       // Index 3
       IF "HMI_Interface_Overview".homeCodition[3].pageIndex = 3 THEN
           "HMI_Interface_Overview".homeCodition[3].emOverviewTitle := WSTRING#'Attachment Home Condition 1';
           "HMI_Interface_Overview".homeCodition[3].emOverviewCmName[0] := WSTRING#'Top Tape X-Axis';
           "HMI_Interface_Overview".homeCodition[3].emOverviewCmName[1] := WSTRING#'Top Tape Attachment';
           "HMI_Interface_Overview".homeCodition[3].emOverviewCmName[2] := WSTRING#'Top Tape Attachment Vacuum';
           "HMI_Interface_Overview".homeCodition[3].emOverviewCmName[3] := WSTRING#'Spare';
           "HMI_Interface_Overview".homeCodition[3].emOverviewCmName[4] := WSTRING#'Spare';
           "HMI_Interface_Overview".homeCodition[3].emOverviewCmName[5] := WSTRING#'Spare';
           "HMI_Interface_Overview".homeCodition[3].emOverviewCmName[6] := WSTRING#'Spare';
           "HMI_Interface_Overview".homeCodition[3].emOverviewCmName[7] := WSTRING#'Spare';
           "HMI_Interface_Overview".homeCodition[3].emOverviewCmName[8] := WSTRING#'Spare';
           "HMI_Interface_Overview".homeCodition[3].emOverviewCmName[9] := WSTRING#'Spare';
           "HMI_Interface_Overview".homeCodition[3].emOverviewCmName[10] := WSTRING#'Spare';
           "HMI_Interface_Overview".homeCodition[3].emOverviewCmName[11] := WSTRING#'Spare';
           "HMI_Interface_Overview".homeCodition[3].emOverviewCmName[12] := WSTRING#'Spare';
           "HMI_Interface_Overview".homeCodition[3].emOverviewCmName[13] := WSTRING#'Spare';
           "HMI_Interface_Overview".homeCodition[3].emOverviewCmPositionName[0] := WSTRING#'Wait Position';
           "HMI_Interface_Overview".homeCodition[3].emOverviewCmPositionName[1] := WSTRING#'Up';
           "HMI_Interface_Overview".homeCodition[3].emOverviewCmPositionName[2] := WSTRING#'On';
           "HMI_Interface_Overview".homeCodition[3].emOverviewCmPositionName[3] := WSTRING#'Spare';
           "HMI_Interface_Overview".homeCodition[3].emOverviewCmPositionName[4] := WSTRING#'Spare';
           "HMI_Interface_Overview".homeCodition[3].emOverviewCmPositionName[5] := WSTRING#'Spare';
           "HMI_Interface_Overview".homeCodition[3].emOverviewCmPositionName[6] := WSTRING#'Spare';
           "HMI_Interface_Overview".homeCodition[3].emOverviewCmPositionName[7] := WSTRING#'Spare';
           "HMI_Interface_Overview".homeCodition[3].emOverviewCmPositionName[8] := WSTRING#'Spare';
           "HMI_Interface_Overview".homeCodition[3].emOverviewCmPositionName[9] := WSTRING#'Spare';
           "HMI_Interface_Overview".homeCodition[3].emOverviewCmPositionName[10] := WSTRING#'Spare';
           "HMI_Interface_Overview".homeCodition[3].emOverviewCmPositionName[11] := WSTRING#'Spare';
           "HMI_Interface_Overview".homeCodition[3].emOverviewCmPositionName[12] := WSTRING#'Spare';
           "HMI_Interface_Overview".homeCodition[3].emOverviewCmPositionName[13] := WSTRING#'Spare';
           IF NOT #statLampControl THEN
               "HMI_Interface_Overview".homeCodition[3].emOverviewHomeLampOn[0] := "Unit1.Em3.HmiInterface".cm.softcam.topTapeAxisX.pos00_wait.inPos;
               "HMI_Interface_Overview".homeCodition[3].emOverviewHomeLampOn[1] := "Unit1.Em3.HmiInterface".cmTopTapeAttachmentUpDown.monitoring.inHomePos;
               "HMI_Interface_Overview".homeCodition[3].emOverviewHomeLampOn[2] := "Unit1.Em3.HmiInterface".cmTopTapeAttachmentVaccumOffOn.monitoring.inWorkPos;
               "HMI_Interface_Overview".homeCodition[3].emOverviewHomeLampOn[3] := FALSE;
               "HMI_Interface_Overview".homeCodition[3].emOverviewHomeLampOn[4] := FALSE;
               "HMI_Interface_Overview".homeCodition[3].emOverviewHomeLampOn[5] := FALSE;
               "HMI_Interface_Overview".homeCodition[3].emOverviewHomeLampOn[6] := FALSE;
               "HMI_Interface_Overview".homeCodition[3].emOverviewHomeLampOn[7] := FALSE;
               "HMI_Interface_Overview".homeCodition[3].emOverviewHomeLampOn[8] := FALSE;
               "HMI_Interface_Overview".homeCodition[3].emOverviewHomeLampOn[9] := FALSE;
               "HMI_Interface_Overview".homeCodition[3].emOverviewHomeLampOn[10] := FALSE;
               "HMI_Interface_Overview".homeCodition[3].emOverviewHomeLampOn[11] := FALSE;
               "HMI_Interface_Overview".homeCodition[3].emOverviewHomeLampOn[12] := FALSE;
               "HMI_Interface_Overview".homeCodition[3].emOverviewHomeLampOn[13] := FALSE;
           END_IF;
       END_IF;

       // Index 4
       IF "HMI_Interface_Overview".homeCodition[3].pageIndex = 4 THEN
           "HMI_Interface_Overview".homeCodition[3].emOverviewTitle := WSTRING#'Fix Stage Home Condition 0';
           "HMI_Interface_Overview".homeCodition[3].emOverviewCmName[0] := WSTRING#'Top Tape Y-Axis';
           "HMI_Interface_Overview".homeCodition[3].emOverviewCmName[1] := WSTRING#'Top Tape Clamp Top Left';
           "HMI_Interface_Overview".homeCodition[3].emOverviewCmName[2] := WSTRING#'Top Tape Clamp Top Center';
           "HMI_Interface_Overview".homeCodition[3].emOverviewCmName[3] := WSTRING#'Top Tape Clamp Top Right';
           "HMI_Interface_Overview".homeCodition[3].emOverviewCmName[4] := WSTRING#'Top Tape Clamp Bottom';
           "HMI_Interface_Overview".homeCodition[3].emOverviewCmName[5] := WSTRING#'Top Tape JR Detect';
           "HMI_Interface_Overview".homeCodition[3].emOverviewCmName[6] := WSTRING#'Spare';
           "HMI_Interface_Overview".homeCodition[3].emOverviewCmName[7] := WSTRING#'Spare';
           "HMI_Interface_Overview".homeCodition[3].emOverviewCmName[8] := WSTRING#'Spare';
           "HMI_Interface_Overview".homeCodition[3].emOverviewCmName[9] := WSTRING#'Spare';
           "HMI_Interface_Overview".homeCodition[3].emOverviewCmName[10] := WSTRING#'Spare';
           "HMI_Interface_Overview".homeCodition[3].emOverviewCmName[11] := WSTRING#'Spare';
           "HMI_Interface_Overview".homeCodition[3].emOverviewCmName[12] := WSTRING#'Spare';
           "HMI_Interface_Overview".homeCodition[3].emOverviewCmName[13] := WSTRING#'Spare';
           "HMI_Interface_Overview".homeCodition[3].emOverviewCmPositionName[0] := WSTRING#'Wait Position';
           "HMI_Interface_Overview".homeCodition[3].emOverviewCmPositionName[1] := WSTRING#'Up';
           "HMI_Interface_Overview".homeCodition[3].emOverviewCmPositionName[2] := WSTRING#'Up';
           "HMI_Interface_Overview".homeCodition[3].emOverviewCmPositionName[3] := WSTRING#'Up';
           "HMI_Interface_Overview".homeCodition[3].emOverviewCmPositionName[4] := WSTRING#'Down';
           "HMI_Interface_Overview".homeCodition[3].emOverviewCmPositionName[5] := WSTRING#'Not Detect';
           "HMI_Interface_Overview".homeCodition[3].emOverviewCmPositionName[6] := WSTRING#'Spare';
           "HMI_Interface_Overview".homeCodition[3].emOverviewCmPositionName[7] := WSTRING#'Spare';
           "HMI_Interface_Overview".homeCodition[3].emOverviewCmPositionName[8] := WSTRING#'Spare';
           "HMI_Interface_Overview".homeCodition[3].emOverviewCmPositionName[9] := WSTRING#'Spare';
           "HMI_Interface_Overview".homeCodition[3].emOverviewCmPositionName[10] := WSTRING#'Spare';
           "HMI_Interface_Overview".homeCodition[3].emOverviewCmPositionName[11] := WSTRING#'Spare';
           "HMI_Interface_Overview".homeCodition[3].emOverviewCmPositionName[12] := WSTRING#'Spare';
           "HMI_Interface_Overview".homeCodition[3].emOverviewCmPositionName[13] := WSTRING#'Spare';
           IF NOT #statLampControl THEN
               "HMI_Interface_Overview".homeCodition[3].emOverviewHomeLampOn[0] := "Unit1.Em3.HmiInterface".cm.softcam.topTapeAxisY.pos00_wait.inPos;
               "HMI_Interface_Overview".homeCodition[3].emOverviewHomeLampOn[1] := "Unit1.Em3.HmiInterface".cmTopTapeClampTopLeftUpDown.monitoring.inHomePos;
               "HMI_Interface_Overview".homeCodition[3].emOverviewHomeLampOn[2] := "Unit1.Em3.HmiInterface".cmTopTapeClampTopCenterUpDown.monitoring.inHomePos;
               "HMI_Interface_Overview".homeCodition[3].emOverviewHomeLampOn[3] := "Unit1.Em3.HmiInterface".cmTopTapeClampTopRightUpDown.monitoring.inHomePos;
               "HMI_Interface_Overview".homeCodition[3].emOverviewHomeLampOn[4] := "Unit1.Em3.HmiInterface".cmTopTapeClampBtmDownUp.monitoring.inHomePos;
               "HMI_Interface_Overview".homeCodition[3].emOverviewHomeLampOn[5] := NOT "Unit1.Em3.HmiInterface".cmTopTapeJRDetect.monitoring.processValue;
               "HMI_Interface_Overview".homeCodition[3].emOverviewHomeLampOn[6] := FALSE;
               "HMI_Interface_Overview".homeCodition[3].emOverviewHomeLampOn[7] := FALSE;
               "HMI_Interface_Overview".homeCodition[3].emOverviewHomeLampOn[8] := FALSE;
               "HMI_Interface_Overview".homeCodition[3].emOverviewHomeLampOn[9] := FALSE;
               "HMI_Interface_Overview".homeCodition[3].emOverviewHomeLampOn[10] := FALSE;
               "HMI_Interface_Overview".homeCodition[3].emOverviewHomeLampOn[11] := FALSE;
               "HMI_Interface_Overview".homeCodition[3].emOverviewHomeLampOn[12] := FALSE;
               "HMI_Interface_Overview".homeCodition[3].emOverviewHomeLampOn[13] := FALSE;
           END_IF;
       END_IF;

       // Index 5
       IF "HMI_Interface_Overview".homeCodition[3].pageIndex = 5 THEN
           "HMI_Interface_Overview".homeCodition[3].emOverviewTitle := WSTRING#'Fix Stage Home Condition 1';
           "HMI_Interface_Overview".homeCodition[3].emOverviewCmName[0] := WSTRING#'Top Tape Y-Axis';
           "HMI_Interface_Overview".homeCodition[3].emOverviewCmName[1] := WSTRING#'Top Tape Clamp Top Left';
           "HMI_Interface_Overview".homeCodition[3].emOverviewCmName[2] := WSTRING#'Top Tape Clamp Top Center';
           "HMI_Interface_Overview".homeCodition[3].emOverviewCmName[3] := WSTRING#'Top Tape Clamp Top Right';
           "HMI_Interface_Overview".homeCodition[3].emOverviewCmName[4] := WSTRING#'Top Tape Clamp Bottom';
           "HMI_Interface_Overview".homeCodition[3].emOverviewCmName[5] := WSTRING#'Top Tape JR Detect';
           "HMI_Interface_Overview".homeCodition[3].emOverviewCmName[6] := WSTRING#'Spare';
           "HMI_Interface_Overview".homeCodition[3].emOverviewCmName[7] := WSTRING#'Spare';
           "HMI_Interface_Overview".homeCodition[3].emOverviewCmName[8] := WSTRING#'Spare';
           "HMI_Interface_Overview".homeCodition[3].emOverviewCmName[9] := WSTRING#'Spare';
           "HMI_Interface_Overview".homeCodition[3].emOverviewCmName[10] := WSTRING#'Spare';
           "HMI_Interface_Overview".homeCodition[3].emOverviewCmName[11] := WSTRING#'Spare';
           "HMI_Interface_Overview".homeCodition[3].emOverviewCmName[12] := WSTRING#'Spare';
           "HMI_Interface_Overview".homeCodition[3].emOverviewCmName[13] := WSTRING#'Spare';
           "HMI_Interface_Overview".homeCodition[3].emOverviewCmPositionName[0] := WSTRING#'Wait Position';
           "HMI_Interface_Overview".homeCodition[3].emOverviewCmPositionName[1] := WSTRING#'Down';
           "HMI_Interface_Overview".homeCodition[3].emOverviewCmPositionName[2] := WSTRING#'Down';
           "HMI_Interface_Overview".homeCodition[3].emOverviewCmPositionName[3] := WSTRING#'Down';
           "HMI_Interface_Overview".homeCodition[3].emOverviewCmPositionName[4] := WSTRING#'Up';
           "HMI_Interface_Overview".homeCodition[3].emOverviewCmPositionName[5] := WSTRING#'Detect';
           "HMI_Interface_Overview".homeCodition[3].emOverviewCmPositionName[6] := WSTRING#'Spare';
           "HMI_Interface_Overview".homeCodition[3].emOverviewCmPositionName[7] := WSTRING#'Spare';
           "HMI_Interface_Overview".homeCodition[3].emOverviewCmPositionName[8] := WSTRING#'Spare';
           "HMI_Interface_Overview".homeCodition[3].emOverviewCmPositionName[9] := WSTRING#'Spare';
           "HMI_Interface_Overview".homeCodition[3].emOverviewCmPositionName[10] := WSTRING#'Spare';
           "HMI_Interface_Overview".homeCodition[3].emOverviewCmPositionName[11] := WSTRING#'Spare';
           "HMI_Interface_Overview".homeCodition[3].emOverviewCmPositionName[12] := WSTRING#'Spare';
           "HMI_Interface_Overview".homeCodition[3].emOverviewCmPositionName[13] := WSTRING#'Spare';
           IF NOT #statLampControl THEN
               "HMI_Interface_Overview".homeCodition[3].emOverviewHomeLampOn[0] := "Unit1.Em3.HmiInterface".cm.softcam.topTapeAxisY.pos00_wait.inPos;
               "HMI_Interface_Overview".homeCodition[3].emOverviewHomeLampOn[1] := "Unit1.Em3.HmiInterface".cmTopTapeClampTopLeftUpDown.monitoring.inWorkPos;
               "HMI_Interface_Overview".homeCodition[3].emOverviewHomeLampOn[2] := "Unit1.Em3.HmiInterface".cmTopTapeClampTopCenterUpDown.monitoring.inWorkPos;
               "HMI_Interface_Overview".homeCodition[3].emOverviewHomeLampOn[3] := "Unit1.Em3.HmiInterface".cmTopTapeClampTopRightUpDown.monitoring.inWorkPos;
               "HMI_Interface_Overview".homeCodition[3].emOverviewHomeLampOn[4] := "Unit1.Em3.HmiInterface".cmTopTapeClampBtmDownUp.monitoring.inWorkPos;
               "HMI_Interface_Overview".homeCodition[3].emOverviewHomeLampOn[5] := "Unit1.Em3.HmiInterface".cmTopTapeJRDetect.monitoring.processValue;
               "HMI_Interface_Overview".homeCodition[3].emOverviewHomeLampOn[6] := FALSE;
               "HMI_Interface_Overview".homeCodition[3].emOverviewHomeLampOn[7] := FALSE;
               "HMI_Interface_Overview".homeCodition[3].emOverviewHomeLampOn[8] := FALSE;
               "HMI_Interface_Overview".homeCodition[3].emOverviewHomeLampOn[9] := FALSE;
               "HMI_Interface_Overview".homeCodition[3].emOverviewHomeLampOn[10] := FALSE;
               "HMI_Interface_Overview".homeCodition[3].emOverviewHomeLampOn[11] := FALSE;
               "HMI_Interface_Overview".homeCodition[3].emOverviewHomeLampOn[12] := FALSE;
               "HMI_Interface_Overview".homeCodition[3].emOverviewHomeLampOn[13] := FALSE;
           END_IF;
       END_IF;

   END_REGION
END_REGION

REGION Network 34 (SCL): Em 4 Page Index Mapping
   REGION Page Index

       // Index 0
       IF "HMI_Interface_Overview".homeCodition[4].pageIndex = 0 THEN
           "HMI_Interface_Overview".homeCodition[4].emOverviewTitle := WSTRING#'Loading Home Condition 0';
           "HMI_Interface_Overview".homeCodition[4].emOverviewCmName[0] := WSTRING#'Side Tape Loading';
           "HMI_Interface_Overview".homeCodition[4].emOverviewCmName[1] := WSTRING#'Side Tape Loading Clamp';
           "HMI_Interface_Overview".homeCodition[4].emOverviewCmName[2] := WSTRING#'Side Tape Cutter';
           "HMI_Interface_Overview".homeCodition[4].emOverviewCmName[3] := WSTRING#'Side Tape Cutter Clamp';
           "HMI_Interface_Overview".homeCodition[4].emOverviewCmName[4] := WSTRING#'Side Tape Tension';
           "HMI_Interface_Overview".homeCodition[4].emOverviewCmName[5] := WSTRING#'Spare';
           "HMI_Interface_Overview".homeCodition[4].emOverviewCmName[6] := WSTRING#'Spare';
           "HMI_Interface_Overview".homeCodition[4].emOverviewCmName[7] := WSTRING#'Spare';
           "HMI_Interface_Overview".homeCodition[4].emOverviewCmName[8] := WSTRING#'Spare';
           "HMI_Interface_Overview".homeCodition[4].emOverviewCmName[9] := WSTRING#'Spare';
           "HMI_Interface_Overview".homeCodition[4].emOverviewCmName[10] := WSTRING#'Spare';
           "HMI_Interface_Overview".homeCodition[4].emOverviewCmName[11] := WSTRING#'Spare';
           "HMI_Interface_Overview".homeCodition[4].emOverviewCmName[12] := WSTRING#'Spare';
           "HMI_Interface_Overview".homeCodition[4].emOverviewCmName[13] := WSTRING#'Spare';
           "HMI_Interface_Overview".homeCodition[4].emOverviewCmPositionName[0] := WSTRING#'Down';
           "HMI_Interface_Overview".homeCodition[4].emOverviewCmPositionName[1] := WSTRING#'Open';
           "HMI_Interface_Overview".homeCodition[4].emOverviewCmPositionName[2] := WSTRING#'Backward';
           "HMI_Interface_Overview".homeCodition[4].emOverviewCmPositionName[3] := WSTRING#'Forward';
           "HMI_Interface_Overview".homeCodition[4].emOverviewCmPositionName[4] := WSTRING#'Backward';
           "HMI_Interface_Overview".homeCodition[4].emOverviewCmPositionName[5] := WSTRING#'Spare';
           "HMI_Interface_Overview".homeCodition[4].emOverviewCmPositionName[6] := WSTRING#'Spare';
           "HMI_Interface_Overview".homeCodition[4].emOverviewCmPositionName[7] := WSTRING#'Spare';
           "HMI_Interface_Overview".homeCodition[4].emOverviewCmPositionName[8] := WSTRING#'Spare';
           "HMI_Interface_Overview".homeCodition[4].emOverviewCmPositionName[9] := WSTRING#'Spare';
           "HMI_Interface_Overview".homeCodition[4].emOverviewCmPositionName[10] := WSTRING#'Spare';
           "HMI_Interface_Overview".homeCodition[4].emOverviewCmPositionName[11] := WSTRING#'Spare';
           "HMI_Interface_Overview".homeCodition[4].emOverviewCmPositionName[12] := WSTRING#'Spare';
           "HMI_Interface_Overview".homeCodition[4].emOverviewCmPositionName[13] := WSTRING#'Spare';
           IF NOT #statLampControl THEN
               "HMI_Interface_Overview".homeCodition[4].emOverviewHomeLampOn[0] := "Unit1.Em4.HmiInterface".cmSideTapeLoadingDownUp.monitoring.inHomePos;
               "HMI_Interface_Overview".homeCodition[4].emOverviewHomeLampOn[1] := "Unit1.Em4.HmiInterface".cmSideTapeLoadingClampOpenClose.monitoring.inHomePos;
               "HMI_Interface_Overview".homeCodition[4].emOverviewHomeLampOn[2] := "Unit1.Em4.HmiInterface".cmSideTapeCutterBwdFwd.monitoring.inHomePos;
               "HMI_Interface_Overview".homeCodition[4].emOverviewHomeLampOn[3] := "Unit1.Em4.HmiInterface".cmSideTapeCutterClampBwdFwd.monitoring.inWorkPos;
               "HMI_Interface_Overview".homeCodition[4].emOverviewHomeLampOn[4] := "Unit1.Em4.HmiInterface".cmSideTapeTensionBwdFwd.monitoring.inHomePos;
               "HMI_Interface_Overview".homeCodition[4].emOverviewHomeLampOn[5] := FALSE;
               "HMI_Interface_Overview".homeCodition[4].emOverviewHomeLampOn[6] := FALSE;
               "HMI_Interface_Overview".homeCodition[4].emOverviewHomeLampOn[7] := FALSE;
               "HMI_Interface_Overview".homeCodition[4].emOverviewHomeLampOn[8] := FALSE;
               "HMI_Interface_Overview".homeCodition[4].emOverviewHomeLampOn[9] := FALSE;
               "HMI_Interface_Overview".homeCodition[4].emOverviewHomeLampOn[10] := FALSE;
               "HMI_Interface_Overview".homeCodition[4].emOverviewHomeLampOn[11] := FALSE;
               "HMI_Interface_Overview".homeCodition[4].emOverviewHomeLampOn[12] := FALSE;
               "HMI_Interface_Overview".homeCodition[4].emOverviewHomeLampOn[13] := FALSE;
           END_IF;
       END_IF;

       // Index 1
       IF "HMI_Interface_Overview".homeCodition[4].pageIndex = 1 THEN
           "HMI_Interface_Overview".homeCodition[4].emOverviewTitle := WSTRING#'Loading Home Condition 1';
           "HMI_Interface_Overview".homeCodition[4].emOverviewCmName[0] := WSTRING#'Side Tape Loading';
           "HMI_Interface_Overview".homeCodition[4].emOverviewCmName[1] := WSTRING#'Side Tape Loading Clamp';
           "HMI_Interface_Overview".homeCodition[4].emOverviewCmName[2] := WSTRING#'Side Tape Cutter';
           "HMI_Interface_Overview".homeCodition[4].emOverviewCmName[3] := WSTRING#'Side Tape Cutter Clamp';
           "HMI_Interface_Overview".homeCodition[4].emOverviewCmName[4] := WSTRING#'Side Tape Tension';
           "HMI_Interface_Overview".homeCodition[4].emOverviewCmName[5] := WSTRING#'Spare';
           "HMI_Interface_Overview".homeCodition[4].emOverviewCmName[6] := WSTRING#'Spare';
           "HMI_Interface_Overview".homeCodition[4].emOverviewCmName[7] := WSTRING#'Spare';
           "HMI_Interface_Overview".homeCodition[4].emOverviewCmName[8] := WSTRING#'Spare';
           "HMI_Interface_Overview".homeCodition[4].emOverviewCmName[9] := WSTRING#'Spare';
           "HMI_Interface_Overview".homeCodition[4].emOverviewCmName[10] := WSTRING#'Spare';
           "HMI_Interface_Overview".homeCodition[4].emOverviewCmName[11] := WSTRING#'Spare';
           "HMI_Interface_Overview".homeCodition[4].emOverviewCmName[12] := WSTRING#'Spare';
           "HMI_Interface_Overview".homeCodition[4].emOverviewCmName[13] := WSTRING#'Spare';
           "HMI_Interface_Overview".homeCodition[4].emOverviewCmPositionName[0] := WSTRING#'Down';
           "HMI_Interface_Overview".homeCodition[4].emOverviewCmPositionName[1] := WSTRING#'Close';
           "HMI_Interface_Overview".homeCodition[4].emOverviewCmPositionName[2] := WSTRING#'Backward';
           "HMI_Interface_Overview".homeCodition[4].emOverviewCmPositionName[3] := WSTRING#'Forward';
           "HMI_Interface_Overview".homeCodition[4].emOverviewCmPositionName[4] := WSTRING#'Backward';
           "HMI_Interface_Overview".homeCodition[4].emOverviewCmPositionName[5] := WSTRING#'Spare';
           "HMI_Interface_Overview".homeCodition[4].emOverviewCmPositionName[6] := WSTRING#'Spare';
           "HMI_Interface_Overview".homeCodition[4].emOverviewCmPositionName[7] := WSTRING#'Spare';
           "HMI_Interface_Overview".homeCodition[4].emOverviewCmPositionName[8] := WSTRING#'Spare';
           "HMI_Interface_Overview".homeCodition[4].emOverviewCmPositionName[9] := WSTRING#'Spare';
           "HMI_Interface_Overview".homeCodition[4].emOverviewCmPositionName[10] := WSTRING#'Spare';
           "HMI_Interface_Overview".homeCodition[4].emOverviewCmPositionName[11] := WSTRING#'Spare';
           "HMI_Interface_Overview".homeCodition[4].emOverviewCmPositionName[12] := WSTRING#'Spare';
           "HMI_Interface_Overview".homeCodition[4].emOverviewCmPositionName[13] := WSTRING#'Spare';
           IF NOT #statLampControl THEN
               "HMI_Interface_Overview".homeCodition[4].emOverviewHomeLampOn[0] := "Unit1.Em4.HmiInterface".cmSideTapeLoadingDownUp.monitoring.inHomePos;
               "HMI_Interface_Overview".homeCodition[4].emOverviewHomeLampOn[1] := "Unit1.Em4.HmiInterface".cmSideTapeLoadingClampOpenClose.monitoring.inWorkPos;
               "HMI_Interface_Overview".homeCodition[4].emOverviewHomeLampOn[2] := "Unit1.Em4.HmiInterface".cmSideTapeCutterBwdFwd.monitoring.inHomePos;
               "HMI_Interface_Overview".homeCodition[4].emOverviewHomeLampOn[3] := "Unit1.Em4.HmiInterface".cmSideTapeCutterClampBwdFwd.monitoring.inWorkPos;
               "HMI_Interface_Overview".homeCodition[4].emOverviewHomeLampOn[4] := "Unit1.Em4.HmiInterface".cmSideTapeTensionBwdFwd.monitoring.inHomePos;
               "HMI_Interface_Overview".homeCodition[4].emOverviewHomeLampOn[5] := FALSE;
               "HMI_Interface_Overview".homeCodition[4].emOverviewHomeLampOn[6] := FALSE;
               "HMI_Interface_Overview".homeCodition[4].emOverviewHomeLampOn[7] := FALSE;
               "HMI_Interface_Overview".homeCodition[4].emOverviewHomeLampOn[8] := FALSE;
               "HMI_Interface_Overview".homeCodition[4].emOverviewHomeLampOn[9] := FALSE;
               "HMI_Interface_Overview".homeCodition[4].emOverviewHomeLampOn[10] := FALSE;
               "HMI_Interface_Overview".homeCodition[4].emOverviewHomeLampOn[11] := FALSE;
               "HMI_Interface_Overview".homeCodition[4].emOverviewHomeLampOn[12] := FALSE;
               "HMI_Interface_Overview".homeCodition[4].emOverviewHomeLampOn[13] := FALSE;
           END_IF;
       END_IF;

       // Index 2
       IF "HMI_Interface_Overview".homeCodition[4].pageIndex = 2 THEN
           "HMI_Interface_Overview".homeCodition[4].emOverviewTitle := WSTRING#'Attachment Home Condition 0';
           "HMI_Interface_Overview".homeCodition[4].emOverviewCmName[0] := WSTRING#'Side Tape Attachment X-Axis';
           "HMI_Interface_Overview".homeCodition[4].emOverviewCmName[1] := WSTRING#'Side Tape Attachment Y-Axis';
           "HMI_Interface_Overview".homeCodition[4].emOverviewCmName[2] := WSTRING#'Side Tape Attachment Left';
           "HMI_Interface_Overview".homeCodition[4].emOverviewCmName[3] := WSTRING#'Side Tape Attachment Right';
           "HMI_Interface_Overview".homeCodition[4].emOverviewCmName[4] := WSTRING#'Side Tape Attachment Bottom';
           "HMI_Interface_Overview".homeCodition[4].emOverviewCmName[5] := WSTRING#'Side Tape Attachment #1 Top Vaccum';
           "HMI_Interface_Overview".homeCodition[4].emOverviewCmName[6] := WSTRING#'Side Tape Attachment #1 Bottom Vaccum';
           "HMI_Interface_Overview".homeCodition[4].emOverviewCmName[7] := WSTRING#'Side Tape Attachment #2 Top Vaccum';
           "HMI_Interface_Overview".homeCodition[4].emOverviewCmName[8] := WSTRING#'Side Tape Attachment #2 Bottom Vaccum';
           "HMI_Interface_Overview".homeCodition[4].emOverviewCmName[9] := WSTRING#'Spare';
           "HMI_Interface_Overview".homeCodition[4].emOverviewCmName[10] := WSTRING#'Spare';
           "HMI_Interface_Overview".homeCodition[4].emOverviewCmName[11] := WSTRING#'Spare';
           "HMI_Interface_Overview".homeCodition[4].emOverviewCmName[12] := WSTRING#'Spare';
           "HMI_Interface_Overview".homeCodition[4].emOverviewCmName[13] := WSTRING#'Spare';
           "HMI_Interface_Overview".homeCodition[4].emOverviewCmPositionName[0] := WSTRING#'Wait Position';
           "HMI_Interface_Overview".homeCodition[4].emOverviewCmPositionName[1] := WSTRING#'Wait Position';
           "HMI_Interface_Overview".homeCodition[4].emOverviewCmPositionName[2] := WSTRING#'Backward';
           "HMI_Interface_Overview".homeCodition[4].emOverviewCmPositionName[3] := WSTRING#'Backward';
           "HMI_Interface_Overview".homeCodition[4].emOverviewCmPositionName[4] := WSTRING#'Forward';
           "HMI_Interface_Overview".homeCodition[4].emOverviewCmPositionName[5] := WSTRING#'Off';
           "HMI_Interface_Overview".homeCodition[4].emOverviewCmPositionName[6] := WSTRING#'Off';
           "HMI_Interface_Overview".homeCodition[4].emOverviewCmPositionName[7] := WSTRING#'Off';
           "HMI_Interface_Overview".homeCodition[4].emOverviewCmPositionName[8] := WSTRING#'Off';
           "HMI_Interface_Overview".homeCodition[4].emOverviewCmPositionName[9] := WSTRING#'Spare';
           "HMI_Interface_Overview".homeCodition[4].emOverviewCmPositionName[10] := WSTRING#'Spare';
           "HMI_Interface_Overview".homeCodition[4].emOverviewCmPositionName[11] := WSTRING#'Spare';
           "HMI_Interface_Overview".homeCodition[4].emOverviewCmPositionName[12] := WSTRING#'Spare';
           "HMI_Interface_Overview".homeCodition[4].emOverviewCmPositionName[13] := WSTRING#'Spare';
           IF NOT #statLampControl THEN
               "HMI_Interface_Overview".homeCodition[4].emOverviewHomeLampOn[0] := "Unit1.Em4.HmiInterface".cm.softcam.sideTapeAttachmentAxisX.pos00_wait.inPos;
               "HMI_Interface_Overview".homeCodition[4].emOverviewHomeLampOn[1] := "Unit1.Em4.HmiInterface".cm.softcam.sideTapeAttachmentAxisY.Pos00_wait.inPos;
               "HMI_Interface_Overview".homeCodition[4].emOverviewHomeLampOn[2] := "Unit1.Em4.HmiInterface".cmSideTapeAttachmentLeftBwdFwd.monitoring.inHomePos;
               "HMI_Interface_Overview".homeCodition[4].emOverviewHomeLampOn[3] := "Unit1.Em4.HmiInterface".cmSideTapeAttachmentRightBwdFwd.monitoring.inHomePos;
               "HMI_Interface_Overview".homeCodition[4].emOverviewHomeLampOn[4] := "Unit1.Em4.HmiInterface".cmSideTapeAttachmentBtmBwdFwd.monitoring.inWorkPos;
               "HMI_Interface_Overview".homeCodition[4].emOverviewHomeLampOn[5] := "Unit1.Em4.HmiInterface".cmSideTapeAttachment1TopVaccumOffOn.monitoring.inHomePos;
               "HMI_Interface_Overview".homeCodition[4].emOverviewHomeLampOn[6] := "Unit1.Em4.HmiInterface".cmSideTapeAttachment1BtmVaccumOffOn.monitoring.inHomePos;
               "HMI_Interface_Overview".homeCodition[4].emOverviewHomeLampOn[7] := "Unit1.Em4.HmiInterface".cmSideTapeAttachment2TopVaccumOffOn.monitoring.inHomePos;
               "HMI_Interface_Overview".homeCodition[4].emOverviewHomeLampOn[8] := "Unit1.Em4.HmiInterface".cmSideTapeAttachment2BtmVaccumOffOn.monitoring.inHomePos;
               "HMI_Interface_Overview".homeCodition[4].emOverviewHomeLampOn[9] := FALSE;
               "HMI_Interface_Overview".homeCodition[4].emOverviewHomeLampOn[10] := FALSE;
               "HMI_Interface_Overview".homeCodition[4].emOverviewHomeLampOn[11] := FALSE;
               "HMI_Interface_Overview".homeCodition[4].emOverviewHomeLampOn[12] := FALSE;
               "HMI_Interface_Overview".homeCodition[4].emOverviewHomeLampOn[13] := FALSE;
           END_IF;
       END_IF;

       // Index 3
       IF "HMI_Interface_Overview".homeCodition[4].pageIndex = 3 THEN
           "HMI_Interface_Overview".homeCodition[4].emOverviewTitle := WSTRING#'Attachment Home Condition 1';
           "HMI_Interface_Overview".homeCodition[4].emOverviewCmName[0] := WSTRING#'Side Tape Attachment X-Axis';
           "HMI_Interface_Overview".homeCodition[4].emOverviewCmName[1] := WSTRING#'Side Tape Attachment Y-Axis';
           "HMI_Interface_Overview".homeCodition[4].emOverviewCmName[2] := WSTRING#'Side Tape Attachment Left';
           "HMI_Interface_Overview".homeCodition[4].emOverviewCmName[3] := WSTRING#'Side Tape Attachment Right';
           "HMI_Interface_Overview".homeCodition[4].emOverviewCmName[4] := WSTRING#'Side Tape Attachment Bottom';
           "HMI_Interface_Overview".homeCodition[4].emOverviewCmName[5] := WSTRING#'Side Tape Attachment #1 Top Vaccum';
           "HMI_Interface_Overview".homeCodition[4].emOverviewCmName[6] := WSTRING#'Side Tape Attachment #1 Bottom Vaccum';
           "HMI_Interface_Overview".homeCodition[4].emOverviewCmName[7] := WSTRING#'Side Tape Attachment #2 Top Vaccum';
           "HMI_Interface_Overview".homeCodition[4].emOverviewCmName[8] := WSTRING#'Side Tape Attachment #2 Bottom Vaccum';
           "HMI_Interface_Overview".homeCodition[4].emOverviewCmName[9] := WSTRING#'Spare';
           "HMI_Interface_Overview".homeCodition[4].emOverviewCmName[10] := WSTRING#'Spare';
           "HMI_Interface_Overview".homeCodition[4].emOverviewCmName[11] := WSTRING#'Spare';
           "HMI_Interface_Overview".homeCodition[4].emOverviewCmName[12] := WSTRING#'Spare';
           "HMI_Interface_Overview".homeCodition[4].emOverviewCmName[13] := WSTRING#'Spare';
           "HMI_Interface_Overview".homeCodition[4].emOverviewCmPositionName[0] := WSTRING#'Wait Position';
           "HMI_Interface_Overview".homeCodition[4].emOverviewCmPositionName[1] := WSTRING#'Wait Position';
           "HMI_Interface_Overview".homeCodition[4].emOverviewCmPositionName[2] := WSTRING#'Backward';
           "HMI_Interface_Overview".homeCodition[4].emOverviewCmPositionName[3] := WSTRING#'Backward';
           "HMI_Interface_Overview".homeCodition[4].emOverviewCmPositionName[4] := WSTRING#'Forward';
           "HMI_Interface_Overview".homeCodition[4].emOverviewCmPositionName[5] := WSTRING#'On';
           "HMI_Interface_Overview".homeCodition[4].emOverviewCmPositionName[6] := WSTRING#'On';
           "HMI_Interface_Overview".homeCodition[4].emOverviewCmPositionName[7] := WSTRING#'Off';
           "HMI_Interface_Overview".homeCodition[4].emOverviewCmPositionName[8] := WSTRING#'Off';
           "HMI_Interface_Overview".homeCodition[4].emOverviewCmPositionName[9] := WSTRING#'Spare';
           "HMI_Interface_Overview".homeCodition[4].emOverviewCmPositionName[10] := WSTRING#'Spare';
           "HMI_Interface_Overview".homeCodition[4].emOverviewCmPositionName[11] := WSTRING#'Spare';
           "HMI_Interface_Overview".homeCodition[4].emOverviewCmPositionName[12] := WSTRING#'Spare';
           "HMI_Interface_Overview".homeCodition[4].emOverviewCmPositionName[13] := WSTRING#'Spare';
           IF NOT #statLampControl THEN
               "HMI_Interface_Overview".homeCodition[4].emOverviewHomeLampOn[0] := "Unit1.Em4.HmiInterface".cm.softcam.sideTapeAttachmentAxisX.pos00_wait.inPos;
               "HMI_Interface_Overview".homeCodition[4].emOverviewHomeLampOn[1] := "Unit1.Em4.HmiInterface".cm.softcam.sideTapeAttachmentAxisY.Pos00_wait.inPos;
               "HMI_Interface_Overview".homeCodition[4].emOverviewHomeLampOn[2] := "Unit1.Em4.HmiInterface".cmSideTapeAttachmentLeftBwdFwd.monitoring.inHomePos;
               "HMI_Interface_Overview".homeCodition[4].emOverviewHomeLampOn[3] := "Unit1.Em4.HmiInterface".cmSideTapeAttachmentRightBwdFwd.monitoring.inHomePos;
               "HMI_Interface_Overview".homeCodition[4].emOverviewHomeLampOn[4] := "Unit1.Em4.HmiInterface".cmSideTapeAttachmentBtmBwdFwd.monitoring.inWorkPos;
               "HMI_Interface_Overview".homeCodition[4].emOverviewHomeLampOn[5] := "Unit1.Em4.HmiInterface".cmSideTapeAttachment1TopVaccumOffOn.monitoring.inWorkPos;
               "HMI_Interface_Overview".homeCodition[4].emOverviewHomeLampOn[6] := "Unit1.Em4.HmiInterface".cmSideTapeAttachment1BtmVaccumOffOn.monitoring.inWorkPos;
               "HMI_Interface_Overview".homeCodition[4].emOverviewHomeLampOn[7] := "Unit1.Em4.HmiInterface".cmSideTapeAttachment2TopVaccumOffOn.monitoring.inHomePos;
               "HMI_Interface_Overview".homeCodition[4].emOverviewHomeLampOn[8] := "Unit1.Em4.HmiInterface".cmSideTapeAttachment2BtmVaccumOffOn.monitoring.inHomePos;
               "HMI_Interface_Overview".homeCodition[4].emOverviewHomeLampOn[9] := FALSE;
               "HMI_Interface_Overview".homeCodition[4].emOverviewHomeLampOn[10] := FALSE;
               "HMI_Interface_Overview".homeCodition[4].emOverviewHomeLampOn[11] := FALSE;
               "HMI_Interface_Overview".homeCodition[4].emOverviewHomeLampOn[12] := FALSE;
               "HMI_Interface_Overview".homeCodition[4].emOverviewHomeLampOn[13] := FALSE;
           END_IF;
       END_IF;

       // Index 4
       IF "HMI_Interface_Overview".homeCodition[4].pageIndex = 4 THEN
           "HMI_Interface_Overview".homeCodition[4].emOverviewTitle := WSTRING#'Attachment Home Condition 2';
           "HMI_Interface_Overview".homeCodition[4].emOverviewCmName[0] := WSTRING#'Side Tape Attachment X-Axis';
           "HMI_Interface_Overview".homeCodition[4].emOverviewCmName[1] := WSTRING#'Side Tape Attachment Y-Axis';
           "HMI_Interface_Overview".homeCodition[4].emOverviewCmName[2] := WSTRING#'Side Tape Attachment Left';
           "HMI_Interface_Overview".homeCodition[4].emOverviewCmName[3] := WSTRING#'Side Tape Attachment Right';
           "HMI_Interface_Overview".homeCodition[4].emOverviewCmName[4] := WSTRING#'Side Tape Attachment Bottom';
           "HMI_Interface_Overview".homeCodition[4].emOverviewCmName[5] := WSTRING#'Side Tape Attachment #1 Top Vaccum';
           "HMI_Interface_Overview".homeCodition[4].emOverviewCmName[6] := WSTRING#'Side Tape Attachment #1 Bottom Vaccum';
           "HMI_Interface_Overview".homeCodition[4].emOverviewCmName[7] := WSTRING#'Side Tape Attachment #2 Top Vaccum';
           "HMI_Interface_Overview".homeCodition[4].emOverviewCmName[8] := WSTRING#'Side Tape Attachment #2 Bottom Vaccum';
           "HMI_Interface_Overview".homeCodition[4].emOverviewCmName[9] := WSTRING#'Spare';
           "HMI_Interface_Overview".homeCodition[4].emOverviewCmName[10] := WSTRING#'Spare';
           "HMI_Interface_Overview".homeCodition[4].emOverviewCmName[11] := WSTRING#'Spare';
           "HMI_Interface_Overview".homeCodition[4].emOverviewCmName[12] := WSTRING#'Spare';
           "HMI_Interface_Overview".homeCodition[4].emOverviewCmName[13] := WSTRING#'Spare';
           "HMI_Interface_Overview".homeCodition[4].emOverviewCmPositionName[0] := WSTRING#'Wait Position';
           "HMI_Interface_Overview".homeCodition[4].emOverviewCmPositionName[1] := WSTRING#'Wait Position';
           "HMI_Interface_Overview".homeCodition[4].emOverviewCmPositionName[2] := WSTRING#'Backward';
           "HMI_Interface_Overview".homeCodition[4].emOverviewCmPositionName[3] := WSTRING#'Backward';
           "HMI_Interface_Overview".homeCodition[4].emOverviewCmPositionName[4] := WSTRING#'Forward';
           "HMI_Interface_Overview".homeCodition[4].emOverviewCmPositionName[5] := WSTRING#'Off';
           "HMI_Interface_Overview".homeCodition[4].emOverviewCmPositionName[6] := WSTRING#'Off';
           "HMI_Interface_Overview".homeCodition[4].emOverviewCmPositionName[7] := WSTRING#'On';
           "HMI_Interface_Overview".homeCodition[4].emOverviewCmPositionName[8] := WSTRING#'On';
           "HMI_Interface_Overview".homeCodition[4].emOverviewCmPositionName[9] := WSTRING#'Spare';
           "HMI_Interface_Overview".homeCodition[4].emOverviewCmPositionName[10] := WSTRING#'Spare';
           "HMI_Interface_Overview".homeCodition[4].emOverviewCmPositionName[11] := WSTRING#'Spare';
           "HMI_Interface_Overview".homeCodition[4].emOverviewCmPositionName[12] := WSTRING#'Spare';
           "HMI_Interface_Overview".homeCodition[4].emOverviewCmPositionName[13] := WSTRING#'Spare';
           IF NOT #statLampControl THEN
               "HMI_Interface_Overview".homeCodition[4].emOverviewHomeLampOn[0] := "Unit1.Em4.HmiInterface".cm.softcam.sideTapeAttachmentAxisX.pos00_wait.inPos;
               "HMI_Interface_Overview".homeCodition[4].emOverviewHomeLampOn[1] := "Unit1.Em4.HmiInterface".cm.softcam.sideTapeAttachmentAxisY.Pos00_wait.inPos;
               "HMI_Interface_Overview".homeCodition[4].emOverviewHomeLampOn[2] := "Unit1.Em4.HmiInterface".cmSideTapeAttachmentLeftBwdFwd.monitoring.inHomePos;
               "HMI_Interface_Overview".homeCodition[4].emOverviewHomeLampOn[3] := "Unit1.Em4.HmiInterface".cmSideTapeAttachmentRightBwdFwd.monitoring.inHomePos;
               "HMI_Interface_Overview".homeCodition[4].emOverviewHomeLampOn[4] := "Unit1.Em4.HmiInterface".cmSideTapeAttachmentBtmBwdFwd.monitoring.inWorkPos;
               "HMI_Interface_Overview".homeCodition[4].emOverviewHomeLampOn[5] := "Unit1.Em4.HmiInterface".cmSideTapeAttachment1TopVaccumOffOn.monitoring.inHomePos;
               "HMI_Interface_Overview".homeCodition[4].emOverviewHomeLampOn[6] := "Unit1.Em4.HmiInterface".cmSideTapeAttachment1BtmVaccumOffOn.monitoring.inHomePos;
               "HMI_Interface_Overview".homeCodition[4].emOverviewHomeLampOn[7] := "Unit1.Em4.HmiInterface".cmSideTapeAttachment2TopVaccumOffOn.monitoring.inWorkPos;
               "HMI_Interface_Overview".homeCodition[4].emOverviewHomeLampOn[8] := "Unit1.Em4.HmiInterface".cmSideTapeAttachment2BtmVaccumOffOn.monitoring.inWorkPos;
               "HMI_Interface_Overview".homeCodition[4].emOverviewHomeLampOn[9] := FALSE;
               "HMI_Interface_Overview".homeCodition[4].emOverviewHomeLampOn[10] := FALSE;
               "HMI_Interface_Overview".homeCodition[4].emOverviewHomeLampOn[11] := FALSE;
               "HMI_Interface_Overview".homeCodition[4].emOverviewHomeLampOn[12] := FALSE;
               "HMI_Interface_Overview".homeCodition[4].emOverviewHomeLampOn[13] := FALSE;
           END_IF;
       END_IF;

       // Index 5
       IF "HMI_Interface_Overview".homeCodition[4].pageIndex = 5 THEN
           "HMI_Interface_Overview".homeCodition[4].emOverviewTitle := WSTRING#'Attachment Home Condition 3';
           "HMI_Interface_Overview".homeCodition[4].emOverviewCmName[0] := WSTRING#'Side Tape Attachment X-Axis';
           "HMI_Interface_Overview".homeCodition[4].emOverviewCmName[1] := WSTRING#'Side Tape Attachment Y-Axis';
           "HMI_Interface_Overview".homeCodition[4].emOverviewCmName[2] := WSTRING#'Side Tape Attachment Left';
           "HMI_Interface_Overview".homeCodition[4].emOverviewCmName[3] := WSTRING#'Side Tape Attachment Right';
           "HMI_Interface_Overview".homeCodition[4].emOverviewCmName[4] := WSTRING#'Side Tape Attachment Bottom';
           "HMI_Interface_Overview".homeCodition[4].emOverviewCmName[5] := WSTRING#'Side Tape Attachment #1 Top Vaccum';
           "HMI_Interface_Overview".homeCodition[4].emOverviewCmName[6] := WSTRING#'Side Tape Attachment #1 Bottom Vaccum';
           "HMI_Interface_Overview".homeCodition[4].emOverviewCmName[7] := WSTRING#'Side Tape Attachment #2 Top Vaccum';
           "HMI_Interface_Overview".homeCodition[4].emOverviewCmName[8] := WSTRING#'Side Tape Attachment #2 Bottom Vaccum';
           "HMI_Interface_Overview".homeCodition[4].emOverviewCmName[9] := WSTRING#'Spare';
           "HMI_Interface_Overview".homeCodition[4].emOverviewCmName[10] := WSTRING#'Spare';
           "HMI_Interface_Overview".homeCodition[4].emOverviewCmName[11] := WSTRING#'Spare';
           "HMI_Interface_Overview".homeCodition[4].emOverviewCmName[12] := WSTRING#'Spare';
           "HMI_Interface_Overview".homeCodition[4].emOverviewCmName[13] := WSTRING#'Spare';
           "HMI_Interface_Overview".homeCodition[4].emOverviewCmPositionName[0] := WSTRING#'Wait Position';
           "HMI_Interface_Overview".homeCodition[4].emOverviewCmPositionName[1] := WSTRING#'Wait Position';
           "HMI_Interface_Overview".homeCodition[4].emOverviewCmPositionName[2] := WSTRING#'Backward';
           "HMI_Interface_Overview".homeCodition[4].emOverviewCmPositionName[3] := WSTRING#'Backward';
           "HMI_Interface_Overview".homeCodition[4].emOverviewCmPositionName[4] := WSTRING#'Forward';
           "HMI_Interface_Overview".homeCodition[4].emOverviewCmPositionName[5] := WSTRING#'On';
           "HMI_Interface_Overview".homeCodition[4].emOverviewCmPositionName[6] := WSTRING#'On';
           "HMI_Interface_Overview".homeCodition[4].emOverviewCmPositionName[7] := WSTRING#'On';
           "HMI_Interface_Overview".homeCodition[4].emOverviewCmPositionName[8] := WSTRING#'On';
           "HMI_Interface_Overview".homeCodition[4].emOverviewCmPositionName[9] := WSTRING#'Spare';
           "HMI_Interface_Overview".homeCodition[4].emOverviewCmPositionName[10] := WSTRING#'Spare';
           "HMI_Interface_Overview".homeCodition[4].emOverviewCmPositionName[11] := WSTRING#'Spare';
           "HMI_Interface_Overview".homeCodition[4].emOverviewCmPositionName[12] := WSTRING#'Spare';
           "HMI_Interface_Overview".homeCodition[4].emOverviewCmPositionName[13] := WSTRING#'Spare';
           IF NOT #statLampControl THEN
               "HMI_Interface_Overview".homeCodition[4].emOverviewHomeLampOn[0] := "Unit1.Em4.HmiInterface".cm.softcam.sideTapeAttachmentAxisX.pos00_wait.inPos;
               "HMI_Interface_Overview".homeCodition[4].emOverviewHomeLampOn[1] := "Unit1.Em4.HmiInterface".cm.softcam.sideTapeAttachmentAxisY.Pos00_wait.inPos;
               "HMI_Interface_Overview".homeCodition[4].emOverviewHomeLampOn[2] := "Unit1.Em4.HmiInterface".cmSideTapeAttachmentLeftBwdFwd.monitoring.inHomePos;
               "HMI_Interface_Overview".homeCodition[4].emOverviewHomeLampOn[3] := "Unit1.Em4.HmiInterface".cmSideTapeAttachmentRightBwdFwd.monitoring.inHomePos;
               "HMI_Interface_Overview".homeCodition[4].emOverviewHomeLampOn[4] := "Unit1.Em4.HmiInterface".cmSideTapeAttachmentBtmBwdFwd.monitoring.inWorkPos;
               "HMI_Interface_Overview".homeCodition[4].emOverviewHomeLampOn[5] := "Unit1.Em4.HmiInterface".cmSideTapeAttachment1TopVaccumOffOn.monitoring.inWorkPos;
               "HMI_Interface_Overview".homeCodition[4].emOverviewHomeLampOn[6] := "Unit1.Em4.HmiInterface".cmSideTapeAttachment1BtmVaccumOffOn.monitoring.inWorkPos;
               "HMI_Interface_Overview".homeCodition[4].emOverviewHomeLampOn[7] := "Unit1.Em4.HmiInterface".cmSideTapeAttachment2TopVaccumOffOn.monitoring.inWorkPos;
               "HMI_Interface_Overview".homeCodition[4].emOverviewHomeLampOn[8] := "Unit1.Em4.HmiInterface".cmSideTapeAttachment2BtmVaccumOffOn.monitoring.inWorkPos;
               "HMI_Interface_Overview".homeCodition[4].emOverviewHomeLampOn[9] := FALSE;
               "HMI_Interface_Overview".homeCodition[4].emOverviewHomeLampOn[10] := FALSE;
               "HMI_Interface_Overview".homeCodition[4].emOverviewHomeLampOn[11] := FALSE;
               "HMI_Interface_Overview".homeCodition[4].emOverviewHomeLampOn[12] := FALSE;
               "HMI_Interface_Overview".homeCodition[4].emOverviewHomeLampOn[13] := FALSE;
           END_IF;
       END_IF;

       // Index 6
       IF "HMI_Interface_Overview".homeCodition[4].pageIndex = 6 THEN
           "HMI_Interface_Overview".homeCodition[4].emOverviewTitle := WSTRING#'Fix Stage Home Condition 0';
           "HMI_Interface_Overview".homeCodition[4].emOverviewCmName[0] := WSTRING#'Side Tape Fix Stage X-Axis';
           "HMI_Interface_Overview".homeCodition[4].emOverviewCmName[1] := WSTRING#'Side Tape Fix Stage C-Axis';
           "HMI_Interface_Overview".homeCodition[4].emOverviewCmName[2] := WSTRING#'Side Tape Fix Stage Clamp';
           "HMI_Interface_Overview".homeCodition[4].emOverviewCmName[3] := WSTRING#'Side Tape Fix Stage JR Detect';
           "HMI_Interface_Overview".homeCodition[4].emOverviewCmName[4] := WSTRING#'Spare';
           "HMI_Interface_Overview".homeCodition[4].emOverviewCmName[5] := WSTRING#'Spare';
           "HMI_Interface_Overview".homeCodition[4].emOverviewCmName[6] := WSTRING#'Spare';
           "HMI_Interface_Overview".homeCodition[4].emOverviewCmName[7] := WSTRING#'Spare';
           "HMI_Interface_Overview".homeCodition[4].emOverviewCmName[8] := WSTRING#'Spare';
           "HMI_Interface_Overview".homeCodition[4].emOverviewCmName[9] := WSTRING#'Spare';
           "HMI_Interface_Overview".homeCodition[4].emOverviewCmName[10] := WSTRING#'Spare';
           "HMI_Interface_Overview".homeCodition[4].emOverviewCmName[11] := WSTRING#'Spare';
           "HMI_Interface_Overview".homeCodition[4].emOverviewCmName[12] := WSTRING#'Spare';
           "HMI_Interface_Overview".homeCodition[4].emOverviewCmName[13] := WSTRING#'Spare';
           "HMI_Interface_Overview".homeCodition[4].emOverviewCmPositionName[0] := WSTRING#'Wait Position';
           "HMI_Interface_Overview".homeCodition[4].emOverviewCmPositionName[1] := WSTRING#'Tape 1 Position';
           "HMI_Interface_Overview".homeCodition[4].emOverviewCmPositionName[2] := WSTRING#'Open';
           "HMI_Interface_Overview".homeCodition[4].emOverviewCmPositionName[3] := WSTRING#'Not Detect';
           "HMI_Interface_Overview".homeCodition[4].emOverviewCmPositionName[4] := WSTRING#'Spare';
           "HMI_Interface_Overview".homeCodition[4].emOverviewCmPositionName[5] := WSTRING#'Spare';
           "HMI_Interface_Overview".homeCodition[4].emOverviewCmPositionName[6] := WSTRING#'Spare';
           "HMI_Interface_Overview".homeCodition[4].emOverviewCmPositionName[7] := WSTRING#'Spare';
           "HMI_Interface_Overview".homeCodition[4].emOverviewCmPositionName[8] := WSTRING#'Spare';
           "HMI_Interface_Overview".homeCodition[4].emOverviewCmPositionName[9] := WSTRING#'Spare';
           "HMI_Interface_Overview".homeCodition[4].emOverviewCmPositionName[10] := WSTRING#'Spare';
           "HMI_Interface_Overview".homeCodition[4].emOverviewCmPositionName[11] := WSTRING#'Spare';
           "HMI_Interface_Overview".homeCodition[4].emOverviewCmPositionName[12] := WSTRING#'Spare';
           "HMI_Interface_Overview".homeCodition[4].emOverviewCmPositionName[13] := WSTRING#'Spare';
           IF NOT #statLampControl THEN
               "HMI_Interface_Overview".homeCodition[4].emOverviewHomeLampOn[0] := "Unit1.Em4.HmiInterface".cm.softcam.sideTapeFixStageAxisX.pos00_wait.inPos;
               "HMI_Interface_Overview".homeCodition[4].emOverviewHomeLampOn[1] := "Unit1.Em4.HmiInterface".cm.softcam.sideTapeFixStageAxisC.pos00_tape1.inPos;
               "HMI_Interface_Overview".homeCodition[4].emOverviewHomeLampOn[2] := "Unit1.Em4.HmiInterface".cmSideTapeFixStageClampOpenClose.monitoring.inHomePos;
               "HMI_Interface_Overview".homeCodition[4].emOverviewHomeLampOn[3] := NOT "Unit1.Em4.HmiInterface".cmSideTapeJRDetect.monitoring.processValue;
               "HMI_Interface_Overview".homeCodition[4].emOverviewHomeLampOn[4] := FALSE;
               "HMI_Interface_Overview".homeCodition[4].emOverviewHomeLampOn[5] := FALSE;
               "HMI_Interface_Overview".homeCodition[4].emOverviewHomeLampOn[6] := FALSE;
               "HMI_Interface_Overview".homeCodition[4].emOverviewHomeLampOn[7] := FALSE;
               "HMI_Interface_Overview".homeCodition[4].emOverviewHomeLampOn[8] := FALSE;
               "HMI_Interface_Overview".homeCodition[4].emOverviewHomeLampOn[9] := FALSE;
               "HMI_Interface_Overview".homeCodition[4].emOverviewHomeLampOn[10] := FALSE;
               "HMI_Interface_Overview".homeCodition[4].emOverviewHomeLampOn[11] := FALSE;
               "HMI_Interface_Overview".homeCodition[4].emOverviewHomeLampOn[12] := FALSE;
               "HMI_Interface_Overview".homeCodition[4].emOverviewHomeLampOn[13] := FALSE;
           END_IF;
       END_IF;

       // Index 7
       IF "HMI_Interface_Overview".homeCodition[4].pageIndex = 7 THEN
           "HMI_Interface_Overview".homeCodition[4].emOverviewTitle := WSTRING#'Fix Stage Home Condition 1';
           "HMI_Interface_Overview".homeCodition[4].emOverviewCmName[0] := WSTRING#'Side Tape Fix Stage X-Axis';
           "HMI_Interface_Overview".homeCodition[4].emOverviewCmName[1] := WSTRING#'Side Tape Fix Stage C-Axis';
           "HMI_Interface_Overview".homeCodition[4].emOverviewCmName[2] := WSTRING#'Side Tape Fix Stage Clamp';
           "HMI_Interface_Overview".homeCodition[4].emOverviewCmName[3] := WSTRING#'Side Tape Fix Stage JR Detect';
           "HMI_Interface_Overview".homeCodition[4].emOverviewCmName[4] := WSTRING#'Spare';
           "HMI_Interface_Overview".homeCodition[4].emOverviewCmName[5] := WSTRING#'Spare';
           "HMI_Interface_Overview".homeCodition[4].emOverviewCmName[6] := WSTRING#'Spare';
           "HMI_Interface_Overview".homeCodition[4].emOverviewCmName[7] := WSTRING#'Spare';
           "HMI_Interface_Overview".homeCodition[4].emOverviewCmName[8] := WSTRING#'Spare';
           "HMI_Interface_Overview".homeCodition[4].emOverviewCmName[9] := WSTRING#'Spare';
           "HMI_Interface_Overview".homeCodition[4].emOverviewCmName[10] := WSTRING#'Spare';
           "HMI_Interface_Overview".homeCodition[4].emOverviewCmName[11] := WSTRING#'Spare';
           "HMI_Interface_Overview".homeCodition[4].emOverviewCmName[12] := WSTRING#'Spare';
           "HMI_Interface_Overview".homeCodition[4].emOverviewCmName[13] := WSTRING#'Spare';
           "HMI_Interface_Overview".homeCodition[4].emOverviewCmPositionName[0] := WSTRING#'Wait Position';
           "HMI_Interface_Overview".homeCodition[4].emOverviewCmPositionName[1] := WSTRING#'Tape 1 Position';
           "HMI_Interface_Overview".homeCodition[4].emOverviewCmPositionName[2] := WSTRING#'Close';
           "HMI_Interface_Overview".homeCodition[4].emOverviewCmPositionName[3] := WSTRING#'Detect';
           "HMI_Interface_Overview".homeCodition[4].emOverviewCmPositionName[4] := WSTRING#'Spare';
           "HMI_Interface_Overview".homeCodition[4].emOverviewCmPositionName[5] := WSTRING#'Spare';
           "HMI_Interface_Overview".homeCodition[4].emOverviewCmPositionName[6] := WSTRING#'Spare';
           "HMI_Interface_Overview".homeCodition[4].emOverviewCmPositionName[7] := WSTRING#'Spare';
           "HMI_Interface_Overview".homeCodition[4].emOverviewCmPositionName[8] := WSTRING#'Spare';
           "HMI_Interface_Overview".homeCodition[4].emOverviewCmPositionName[9] := WSTRING#'Spare';
           "HMI_Interface_Overview".homeCodition[4].emOverviewCmPositionName[10] := WSTRING#'Spare';
           "HMI_Interface_Overview".homeCodition[4].emOverviewCmPositionName[11] := WSTRING#'Spare';
           "HMI_Interface_Overview".homeCodition[4].emOverviewCmPositionName[12] := WSTRING#'Spare';
           "HMI_Interface_Overview".homeCodition[4].emOverviewCmPositionName[13] := WSTRING#'Spare';
           IF NOT #statLampControl THEN
               "HMI_Interface_Overview".homeCodition[4].emOverviewHomeLampOn[0] := "Unit1.Em4.HmiInterface".cm.softcam.sideTapeFixStageAxisX.pos00_wait.inPos;
               "HMI_Interface_Overview".homeCodition[4].emOverviewHomeLampOn[1] := "Unit1.Em4.HmiInterface".cm.softcam.sideTapeFixStageAxisC.pos00_tape1.inPos;
               "HMI_Interface_Overview".homeCodition[4].emOverviewHomeLampOn[2] := "Unit1.Em4.HmiInterface".cmSideTapeFixStageClampOpenClose.monitoring.inWorkPos;
               "HMI_Interface_Overview".homeCodition[4].emOverviewHomeLampOn[3] := "Unit1.Em4.HmiInterface".cmSideTapeJRDetect.monitoring.processValue;
               "HMI_Interface_Overview".homeCodition[4].emOverviewHomeLampOn[4] := FALSE;
               "HMI_Interface_Overview".homeCodition[4].emOverviewHomeLampOn[5] := FALSE;
               "HMI_Interface_Overview".homeCodition[4].emOverviewHomeLampOn[6] := FALSE;
               "HMI_Interface_Overview".homeCodition[4].emOverviewHomeLampOn[7] := FALSE;
               "HMI_Interface_Overview".homeCodition[4].emOverviewHomeLampOn[8] := FALSE;
               "HMI_Interface_Overview".homeCodition[4].emOverviewHomeLampOn[9] := FALSE;
               "HMI_Interface_Overview".homeCodition[4].emOverviewHomeLampOn[10] := FALSE;
               "HMI_Interface_Overview".homeCodition[4].emOverviewHomeLampOn[11] := FALSE;
               "HMI_Interface_Overview".homeCodition[4].emOverviewHomeLampOn[12] := FALSE;
               "HMI_Interface_Overview".homeCodition[4].emOverviewHomeLampOn[13] := FALSE;
           END_IF;
       END_IF;

       // Index 8
       IF "HMI_Interface_Overview".homeCodition[4].pageIndex = 8 THEN
           "HMI_Interface_Overview".homeCodition[4].emOverviewTitle := WSTRING#'Fix Stage Home Condition 2';
           "HMI_Interface_Overview".homeCodition[4].emOverviewCmName[0] := WSTRING#'Side Tape Fix Stage X-Axis';
           "HMI_Interface_Overview".homeCodition[4].emOverviewCmName[1] := WSTRING#'Side Tape Fix Stage C-Axis';
           "HMI_Interface_Overview".homeCodition[4].emOverviewCmName[2] := WSTRING#'Side Tape Fix Stage Clamp';
           "HMI_Interface_Overview".homeCodition[4].emOverviewCmName[3] := WSTRING#'Side Tape Fix Stage JR Detect';
           "HMI_Interface_Overview".homeCodition[4].emOverviewCmName[4] := WSTRING#'Spare';
           "HMI_Interface_Overview".homeCodition[4].emOverviewCmName[5] := WSTRING#'Spare';
           "HMI_Interface_Overview".homeCodition[4].emOverviewCmName[6] := WSTRING#'Spare';
           "HMI_Interface_Overview".homeCodition[4].emOverviewCmName[7] := WSTRING#'Spare';
           "HMI_Interface_Overview".homeCodition[4].emOverviewCmName[8] := WSTRING#'Spare';
           "HMI_Interface_Overview".homeCodition[4].emOverviewCmName[9] := WSTRING#'Spare';
           "HMI_Interface_Overview".homeCodition[4].emOverviewCmName[10] := WSTRING#'Spare';
           "HMI_Interface_Overview".homeCodition[4].emOverviewCmName[11] := WSTRING#'Spare';
           "HMI_Interface_Overview".homeCodition[4].emOverviewCmName[12] := WSTRING#'Spare';
           "HMI_Interface_Overview".homeCodition[4].emOverviewCmName[13] := WSTRING#'Spare';
           "HMI_Interface_Overview".homeCodition[4].emOverviewCmPositionName[0] := WSTRING#'Wait Position';
           "HMI_Interface_Overview".homeCodition[4].emOverviewCmPositionName[1] := WSTRING#'Tape 2 Position';
           "HMI_Interface_Overview".homeCodition[4].emOverviewCmPositionName[2] := WSTRING#'Close';
           "HMI_Interface_Overview".homeCodition[4].emOverviewCmPositionName[3] := WSTRING#'Detect';
           "HMI_Interface_Overview".homeCodition[4].emOverviewCmPositionName[4] := WSTRING#'Spare';
           "HMI_Interface_Overview".homeCodition[4].emOverviewCmPositionName[5] := WSTRING#'Spare';
           "HMI_Interface_Overview".homeCodition[4].emOverviewCmPositionName[6] := WSTRING#'Spare';
           "HMI_Interface_Overview".homeCodition[4].emOverviewCmPositionName[7] := WSTRING#'Spare';
           "HMI_Interface_Overview".homeCodition[4].emOverviewCmPositionName[8] := WSTRING#'Spare';
           "HMI_Interface_Overview".homeCodition[4].emOverviewCmPositionName[9] := WSTRING#'Spare';
           "HMI_Interface_Overview".homeCodition[4].emOverviewCmPositionName[10] := WSTRING#'Spare';
           "HMI_Interface_Overview".homeCodition[4].emOverviewCmPositionName[11] := WSTRING#'Spare';
           "HMI_Interface_Overview".homeCodition[4].emOverviewCmPositionName[12] := WSTRING#'Spare';
           "HMI_Interface_Overview".homeCodition[4].emOverviewCmPositionName[13] := WSTRING#'Spare';
           IF NOT #statLampControl THEN
               "HMI_Interface_Overview".homeCodition[4].emOverviewHomeLampOn[0] := "Unit1.Em4.HmiInterface".cm.softcam.sideTapeFixStageAxisX.pos00_wait.inPos;
               "HMI_Interface_Overview".homeCodition[4].emOverviewHomeLampOn[1] := "Unit1.Em4.HmiInterface".cm.softcam.sideTapeFixStageAxisC.pos01_tape2.inPos;
               "HMI_Interface_Overview".homeCodition[4].emOverviewHomeLampOn[2] := "Unit1.Em4.HmiInterface".cmSideTapeFixStageClampOpenClose.monitoring.inWorkPos;
               "HMI_Interface_Overview".homeCodition[4].emOverviewHomeLampOn[3] := "Unit1.Em4.HmiInterface".cmSideTapeJRDetect.monitoring.processValue;
               "HMI_Interface_Overview".homeCodition[4].emOverviewHomeLampOn[4] := FALSE;
               "HMI_Interface_Overview".homeCodition[4].emOverviewHomeLampOn[5] := FALSE;
               "HMI_Interface_Overview".homeCodition[4].emOverviewHomeLampOn[6] := FALSE;
               "HMI_Interface_Overview".homeCodition[4].emOverviewHomeLampOn[7] := FALSE;
               "HMI_Interface_Overview".homeCodition[4].emOverviewHomeLampOn[8] := FALSE;
               "HMI_Interface_Overview".homeCodition[4].emOverviewHomeLampOn[9] := FALSE;
               "HMI_Interface_Overview".homeCodition[4].emOverviewHomeLampOn[10] := FALSE;
               "HMI_Interface_Overview".homeCodition[4].emOverviewHomeLampOn[11] := FALSE;
               "HMI_Interface_Overview".homeCodition[4].emOverviewHomeLampOn[12] := FALSE;
               "HMI_Interface_Overview".homeCodition[4].emOverviewHomeLampOn[13] := FALSE;
           END_IF;
       END_IF;

       // Index 9
       IF "HMI_Interface_Overview".homeCodition[4].pageIndex = 9 THEN
           "HMI_Interface_Overview".homeCodition[4].emOverviewTitle := WSTRING#'Fix Stage Home Condition 3';
           "HMI_Interface_Overview".homeCodition[4].emOverviewCmName[0] := WSTRING#'Side Tape Fix Stage X-Axis';
           "HMI_Interface_Overview".homeCodition[4].emOverviewCmName[1] := WSTRING#'Side Tape Fix Stage C-Axis';
           "HMI_Interface_Overview".homeCodition[4].emOverviewCmName[2] := WSTRING#'Side Tape Fix Stage Clamp';
           "HMI_Interface_Overview".homeCodition[4].emOverviewCmName[3] := WSTRING#'Side Tape Fix Stage JR Detect';
           "HMI_Interface_Overview".homeCodition[4].emOverviewCmName[4] := WSTRING#'Spare';
           "HMI_Interface_Overview".homeCodition[4].emOverviewCmName[5] := WSTRING#'Spare';
           "HMI_Interface_Overview".homeCodition[4].emOverviewCmName[6] := WSTRING#'Spare';
           "HMI_Interface_Overview".homeCodition[4].emOverviewCmName[7] := WSTRING#'Spare';
           "HMI_Interface_Overview".homeCodition[4].emOverviewCmName[8] := WSTRING#'Spare';
           "HMI_Interface_Overview".homeCodition[4].emOverviewCmName[9] := WSTRING#'Spare';
           "HMI_Interface_Overview".homeCodition[4].emOverviewCmName[10] := WSTRING#'Spare';
           "HMI_Interface_Overview".homeCodition[4].emOverviewCmName[11] := WSTRING#'Spare';
           "HMI_Interface_Overview".homeCodition[4].emOverviewCmName[12] := WSTRING#'Spare';
           "HMI_Interface_Overview".homeCodition[4].emOverviewCmName[13] := WSTRING#'Spare';
           "HMI_Interface_Overview".homeCodition[4].emOverviewCmPositionName[0] := WSTRING#'Wait Position';
           "HMI_Interface_Overview".homeCodition[4].emOverviewCmPositionName[1] := WSTRING#'Tape 3 Position';
           "HMI_Interface_Overview".homeCodition[4].emOverviewCmPositionName[2] := WSTRING#'Close';
           "HMI_Interface_Overview".homeCodition[4].emOverviewCmPositionName[3] := WSTRING#'Detect';
           "HMI_Interface_Overview".homeCodition[4].emOverviewCmPositionName[4] := WSTRING#'Spare';
           "HMI_Interface_Overview".homeCodition[4].emOverviewCmPositionName[5] := WSTRING#'Spare';
           "HMI_Interface_Overview".homeCodition[4].emOverviewCmPositionName[6] := WSTRING#'Spare';
           "HMI_Interface_Overview".homeCodition[4].emOverviewCmPositionName[7] := WSTRING#'Spare';
           "HMI_Interface_Overview".homeCodition[4].emOverviewCmPositionName[8] := WSTRING#'Spare';
           "HMI_Interface_Overview".homeCodition[4].emOverviewCmPositionName[9] := WSTRING#'Spare';
           "HMI_Interface_Overview".homeCodition[4].emOverviewCmPositionName[10] := WSTRING#'Spare';
           "HMI_Interface_Overview".homeCodition[4].emOverviewCmPositionName[11] := WSTRING#'Spare';
           "HMI_Interface_Overview".homeCodition[4].emOverviewCmPositionName[12] := WSTRING#'Spare';
           "HMI_Interface_Overview".homeCodition[4].emOverviewCmPositionName[13] := WSTRING#'Spare';
           IF NOT #statLampControl THEN
               "HMI_Interface_Overview".homeCodition[4].emOverviewHomeLampOn[0] := "Unit1.Em4.HmiInterface".cm.softcam.sideTapeFixStageAxisX.pos00_wait.inPos;
               "HMI_Interface_Overview".homeCodition[4].emOverviewHomeLampOn[1] := "Unit1.Em4.HmiInterface".cm.softcam.sideTapeFixStageAxisC.pos02_tape3.inPos;
               "HMI_Interface_Overview".homeCodition[4].emOverviewHomeLampOn[2] := "Unit1.Em4.HmiInterface".cmSideTapeFixStageClampOpenClose.monitoring.inWorkPos;
               "HMI_Interface_Overview".homeCodition[4].emOverviewHomeLampOn[3] := "Unit1.Em4.HmiInterface".cmSideTapeJRDetect.monitoring.processValue;
               "HMI_Interface_Overview".homeCodition[4].emOverviewHomeLampOn[4] := FALSE;
               "HMI_Interface_Overview".homeCodition[4].emOverviewHomeLampOn[5] := FALSE;
               "HMI_Interface_Overview".homeCodition[4].emOverviewHomeLampOn[6] := FALSE;
               "HMI_Interface_Overview".homeCodition[4].emOverviewHomeLampOn[7] := FALSE;
               "HMI_Interface_Overview".homeCodition[4].emOverviewHomeLampOn[8] := FALSE;
               "HMI_Interface_Overview".homeCodition[4].emOverviewHomeLampOn[9] := FALSE;
               "HMI_Interface_Overview".homeCodition[4].emOverviewHomeLampOn[10] := FALSE;
               "HMI_Interface_Overview".homeCodition[4].emOverviewHomeLampOn[11] := FALSE;
               "HMI_Interface_Overview".homeCodition[4].emOverviewHomeLampOn[12] := FALSE;
               "HMI_Interface_Overview".homeCodition[4].emOverviewHomeLampOn[13] := FALSE;
           END_IF;
       END_IF;

       // Index 10
       IF "HMI_Interface_Overview".homeCodition[4].pageIndex = 10 THEN
           "HMI_Interface_Overview".homeCodition[4].emOverviewTitle := WSTRING#'Fix Stage Home Condition 4';
           "HMI_Interface_Overview".homeCodition[4].emOverviewCmName[0] := WSTRING#'Side Tape Fix Stage X-Axis';
           "HMI_Interface_Overview".homeCodition[4].emOverviewCmName[1] := WSTRING#'Side Tape Fix Stage C-Axis';
           "HMI_Interface_Overview".homeCodition[4].emOverviewCmName[2] := WSTRING#'Side Tape Fix Stage Clamp';
           "HMI_Interface_Overview".homeCodition[4].emOverviewCmName[3] := WSTRING#'Side Tape Fix Stage JR Detect';
           "HMI_Interface_Overview".homeCodition[4].emOverviewCmName[4] := WSTRING#'Spare';
           "HMI_Interface_Overview".homeCodition[4].emOverviewCmName[5] := WSTRING#'Spare';
           "HMI_Interface_Overview".homeCodition[4].emOverviewCmName[6] := WSTRING#'Spare';
           "HMI_Interface_Overview".homeCodition[4].emOverviewCmName[7] := WSTRING#'Spare';
           "HMI_Interface_Overview".homeCodition[4].emOverviewCmName[8] := WSTRING#'Spare';
           "HMI_Interface_Overview".homeCodition[4].emOverviewCmName[9] := WSTRING#'Spare';
           "HMI_Interface_Overview".homeCodition[4].emOverviewCmName[10] := WSTRING#'Spare';
           "HMI_Interface_Overview".homeCodition[4].emOverviewCmName[11] := WSTRING#'Spare';
           "HMI_Interface_Overview".homeCodition[4].emOverviewCmName[12] := WSTRING#'Spare';
           "HMI_Interface_Overview".homeCodition[4].emOverviewCmName[13] := WSTRING#'Spare';
           "HMI_Interface_Overview".homeCodition[4].emOverviewCmPositionName[0] := WSTRING#'Wait Position';
           "HMI_Interface_Overview".homeCodition[4].emOverviewCmPositionName[1] := WSTRING#'Tape 4 Position';
           "HMI_Interface_Overview".homeCodition[4].emOverviewCmPositionName[2] := WSTRING#'Close';
           "HMI_Interface_Overview".homeCodition[4].emOverviewCmPositionName[3] := WSTRING#'Detect';
           "HMI_Interface_Overview".homeCodition[4].emOverviewCmPositionName[4] := WSTRING#'Spare';
           "HMI_Interface_Overview".homeCodition[4].emOverviewCmPositionName[5] := WSTRING#'Spare';
           "HMI_Interface_Overview".homeCodition[4].emOverviewCmPositionName[6] := WSTRING#'Spare';
           "HMI_Interface_Overview".homeCodition[4].emOverviewCmPositionName[7] := WSTRING#'Spare';
           "HMI_Interface_Overview".homeCodition[4].emOverviewCmPositionName[8] := WSTRING#'Spare';
           "HMI_Interface_Overview".homeCodition[4].emOverviewCmPositionName[9] := WSTRING#'Spare';
           "HMI_Interface_Overview".homeCodition[4].emOverviewCmPositionName[10] := WSTRING#'Spare';
           "HMI_Interface_Overview".homeCodition[4].emOverviewCmPositionName[11] := WSTRING#'Spare';
           "HMI_Interface_Overview".homeCodition[4].emOverviewCmPositionName[12] := WSTRING#'Spare';
           "HMI_Interface_Overview".homeCodition[4].emOverviewCmPositionName[13] := WSTRING#'Spare';
           IF NOT #statLampControl THEN
               "HMI_Interface_Overview".homeCodition[4].emOverviewHomeLampOn[0] := "Unit1.Em4.HmiInterface".cm.softcam.sideTapeFixStageAxisX.pos00_wait.inPos;
               "HMI_Interface_Overview".homeCodition[4].emOverviewHomeLampOn[1] := "Unit1.Em4.HmiInterface".cm.softcam.sideTapeFixStageAxisC.pos03_tape4.inPos;
               "HMI_Interface_Overview".homeCodition[4].emOverviewHomeLampOn[2] := "Unit1.Em4.HmiInterface".cmSideTapeFixStageClampOpenClose.monitoring.inWorkPos;
               "HMI_Interface_Overview".homeCodition[4].emOverviewHomeLampOn[3] := "Unit1.Em4.HmiInterface".cmSideTapeJRDetect.monitoring.processValue;
               "HMI_Interface_Overview".homeCodition[4].emOverviewHomeLampOn[4] := FALSE;
               "HMI_Interface_Overview".homeCodition[4].emOverviewHomeLampOn[5] := FALSE;
               "HMI_Interface_Overview".homeCodition[4].emOverviewHomeLampOn[6] := FALSE;
               "HMI_Interface_Overview".homeCodition[4].emOverviewHomeLampOn[7] := FALSE;
               "HMI_Interface_Overview".homeCodition[4].emOverviewHomeLampOn[8] := FALSE;
               "HMI_Interface_Overview".homeCodition[4].emOverviewHomeLampOn[9] := FALSE;
               "HMI_Interface_Overview".homeCodition[4].emOverviewHomeLampOn[10] := FALSE;
               "HMI_Interface_Overview".homeCodition[4].emOverviewHomeLampOn[11] := FALSE;
               "HMI_Interface_Overview".homeCodition[4].emOverviewHomeLampOn[12] := FALSE;
               "HMI_Interface_Overview".homeCodition[4].emOverviewHomeLampOn[13] := FALSE;
           END_IF;
       END_IF;

   END_REGION
END_REGION

REGION Network 35 (SCL): Em 5 Page Index Mapping
   REGION Page Index

       // Index 0
       IF "HMI_Interface_Overview".homeCodition[5].pageIndex = 0 THEN
           "HMI_Interface_Overview".homeCodition[5].emOverviewTitle := WSTRING#'P&P Left Home Condition 0';
           "HMI_Interface_Overview".homeCodition[5].emOverviewCmName[0] := WSTRING#'Transfer P&P Left X-Axis';
           "HMI_Interface_Overview".homeCodition[5].emOverviewCmName[1] := WSTRING#'Transfer P&P Left Y-Axis';
           "HMI_Interface_Overview".homeCodition[5].emOverviewCmName[2] := WSTRING#'Transfer P&P Left Z-Axis';
           "HMI_Interface_Overview".homeCodition[5].emOverviewCmName[3] := WSTRING#'Transfer P&P Left Clamp';
           "HMI_Interface_Overview".homeCodition[5].emOverviewCmName[4] := WSTRING#'Transfer P&P Left JR Detect';
           "HMI_Interface_Overview".homeCodition[5].emOverviewCmName[5] := WSTRING#'Spare';
           "HMI_Interface_Overview".homeCodition[5].emOverviewCmName[6] := WSTRING#'Spare';
           "HMI_Interface_Overview".homeCodition[5].emOverviewCmName[7] := WSTRING#'Spare';
           "HMI_Interface_Overview".homeCodition[5].emOverviewCmName[8] := WSTRING#'Spare';
           "HMI_Interface_Overview".homeCodition[5].emOverviewCmName[9] := WSTRING#'Spare';
           "HMI_Interface_Overview".homeCodition[5].emOverviewCmName[10] := WSTRING#'Spare';
           "HMI_Interface_Overview".homeCodition[5].emOverviewCmName[11] := WSTRING#'Spare';
           "HMI_Interface_Overview".homeCodition[5].emOverviewCmName[12] := WSTRING#'Spare';
           "HMI_Interface_Overview".homeCodition[5].emOverviewCmName[13] := WSTRING#'Spare';
           "HMI_Interface_Overview".homeCodition[5].emOverviewCmPositionName[0] := WSTRING#'Wait Position';
           "HMI_Interface_Overview".homeCodition[5].emOverviewCmPositionName[1] := WSTRING#'Wait Position';
           "HMI_Interface_Overview".homeCodition[5].emOverviewCmPositionName[2] := WSTRING#'Wait Position';
           "HMI_Interface_Overview".homeCodition[5].emOverviewCmPositionName[3] := WSTRING#'Open';
           "HMI_Interface_Overview".homeCodition[5].emOverviewCmPositionName[4] := WSTRING#'Not Detect';
           "HMI_Interface_Overview".homeCodition[5].emOverviewCmPositionName[5] := WSTRING#'Spare';
           "HMI_Interface_Overview".homeCodition[5].emOverviewCmPositionName[6] := WSTRING#'Spare';
           "HMI_Interface_Overview".homeCodition[5].emOverviewCmPositionName[7] := WSTRING#'Spare';
           "HMI_Interface_Overview".homeCodition[5].emOverviewCmPositionName[8] := WSTRING#'Spare';
           "HMI_Interface_Overview".homeCodition[5].emOverviewCmPositionName[9] := WSTRING#'Spare';
           "HMI_Interface_Overview".homeCodition[5].emOverviewCmPositionName[10] := WSTRING#'Spare';
           "HMI_Interface_Overview".homeCodition[5].emOverviewCmPositionName[11] := WSTRING#'Spare';
           "HMI_Interface_Overview".homeCodition[5].emOverviewCmPositionName[12] := WSTRING#'Spare';
           "HMI_Interface_Overview".homeCodition[5].emOverviewCmPositionName[13] := WSTRING#'Spare';
           IF NOT #statLampControl THEN
               "HMI_Interface_Overview".homeCodition[5].emOverviewHomeLampOn[0] := "Unit1.Em5.HmiInterface".cm.softcam.transferPnPLeftAxisX.pos00_wait.inPos;
               "HMI_Interface_Overview".homeCodition[5].emOverviewHomeLampOn[1] := "Unit1.Em5.HmiInterface".cm.softcam.transferPnPLeftAxisY.pos00_wait.inPos;
               "HMI_Interface_Overview".homeCodition[5].emOverviewHomeLampOn[2] := "Unit1.Em5.HmiInterface".cm.softcam.transferPnPLeftAxisZ.pos00_wait.inPos;
               "HMI_Interface_Overview".homeCodition[5].emOverviewHomeLampOn[3] := "Unit1.Em5.HmiInterface".cmTransferPnPLeftClampOpenClose.monitoring.inHomePos;
               "HMI_Interface_Overview".homeCodition[5].emOverviewHomeLampOn[4] := NOT "Unit1.Em5.HmiInterface".cmTransferPnPLeftJRDetect.monitoring.processValue;
               "HMI_Interface_Overview".homeCodition[5].emOverviewHomeLampOn[5] := FALSE;
               "HMI_Interface_Overview".homeCodition[5].emOverviewHomeLampOn[6] := FALSE;
               "HMI_Interface_Overview".homeCodition[5].emOverviewHomeLampOn[7] := FALSE;
               "HMI_Interface_Overview".homeCodition[5].emOverviewHomeLampOn[8] := FALSE;
               "HMI_Interface_Overview".homeCodition[5].emOverviewHomeLampOn[9] := FALSE;
               "HMI_Interface_Overview".homeCodition[5].emOverviewHomeLampOn[10] := FALSE;
               "HMI_Interface_Overview".homeCodition[5].emOverviewHomeLampOn[11] := FALSE;
               "HMI_Interface_Overview".homeCodition[5].emOverviewHomeLampOn[12] := FALSE;
               "HMI_Interface_Overview".homeCodition[5].emOverviewHomeLampOn[13] := FALSE;
           END_IF;
       END_IF;

       // Index 1
       IF "HMI_Interface_Overview".homeCodition[5].pageIndex = 1 THEN
           "HMI_Interface_Overview".homeCodition[5].emOverviewTitle := WSTRING#'P&P Left Home Condition 1';
           "HMI_Interface_Overview".homeCodition[5].emOverviewCmName[0] := WSTRING#'Transfer P&P Left X-Axis';
           "HMI_Interface_Overview".homeCodition[5].emOverviewCmName[1] := WSTRING#'Transfer P&P Left Y-Axis';
           "HMI_Interface_Overview".homeCodition[5].emOverviewCmName[2] := WSTRING#'Transfer P&P Left Z-Axis';
           "HMI_Interface_Overview".homeCodition[5].emOverviewCmName[3] := WSTRING#'Transfer P&P Left Clamp';
           "HMI_Interface_Overview".homeCodition[5].emOverviewCmName[4] := WSTRING#'Transfer P&P Left JR Detect';
           "HMI_Interface_Overview".homeCodition[5].emOverviewCmName[5] := WSTRING#'Spare';
           "HMI_Interface_Overview".homeCodition[5].emOverviewCmName[6] := WSTRING#'Spare';
           "HMI_Interface_Overview".homeCodition[5].emOverviewCmName[7] := WSTRING#'Spare';
           "HMI_Interface_Overview".homeCodition[5].emOverviewCmName[8] := WSTRING#'Spare';
           "HMI_Interface_Overview".homeCodition[5].emOverviewCmName[9] := WSTRING#'Spare';
           "HMI_Interface_Overview".homeCodition[5].emOverviewCmName[10] := WSTRING#'Spare';
           "HMI_Interface_Overview".homeCodition[5].emOverviewCmName[11] := WSTRING#'Spare';
           "HMI_Interface_Overview".homeCodition[5].emOverviewCmName[12] := WSTRING#'Spare';
           "HMI_Interface_Overview".homeCodition[5].emOverviewCmName[13] := WSTRING#'Spare';
           "HMI_Interface_Overview".homeCodition[5].emOverviewCmPositionName[0] := WSTRING#'Wait Position';
           "HMI_Interface_Overview".homeCodition[5].emOverviewCmPositionName[1] := WSTRING#'Wait Position';
           "HMI_Interface_Overview".homeCodition[5].emOverviewCmPositionName[2] := WSTRING#'Wait Position';
           "HMI_Interface_Overview".homeCodition[5].emOverviewCmPositionName[3] := WSTRING#'Close';
           "HMI_Interface_Overview".homeCodition[5].emOverviewCmPositionName[4] := WSTRING#'Detect';
           "HMI_Interface_Overview".homeCodition[5].emOverviewCmPositionName[5] := WSTRING#'Spare';
           "HMI_Interface_Overview".homeCodition[5].emOverviewCmPositionName[6] := WSTRING#'Spare';
           "HMI_Interface_Overview".homeCodition[5].emOverviewCmPositionName[7] := WSTRING#'Spare';
           "HMI_Interface_Overview".homeCodition[5].emOverviewCmPositionName[8] := WSTRING#'Spare';
           "HMI_Interface_Overview".homeCodition[5].emOverviewCmPositionName[9] := WSTRING#'Spare';
           "HMI_Interface_Overview".homeCodition[5].emOverviewCmPositionName[10] := WSTRING#'Spare';
           "HMI_Interface_Overview".homeCodition[5].emOverviewCmPositionName[11] := WSTRING#'Spare';
           "HMI_Interface_Overview".homeCodition[5].emOverviewCmPositionName[12] := WSTRING#'Spare';
           "HMI_Interface_Overview".homeCodition[5].emOverviewCmPositionName[13] := WSTRING#'Spare';
           IF NOT #statLampControl THEN
               "HMI_Interface_Overview".homeCodition[5].emOverviewHomeLampOn[0] := "Unit1.Em5.HmiInterface".cm.softcam.transferPnPLeftAxisX.pos00_wait.inPos;
               "HMI_Interface_Overview".homeCodition[5].emOverviewHomeLampOn[1] := "Unit1.Em5.HmiInterface".cm.softcam.transferPnPLeftAxisY.pos00_wait.inPos;
               "HMI_Interface_Overview".homeCodition[5].emOverviewHomeLampOn[2] := "Unit1.Em5.HmiInterface".cm.softcam.transferPnPLeftAxisZ.pos00_wait.inPos;
               "HMI_Interface_Overview".homeCodition[5].emOverviewHomeLampOn[3] := "Unit1.Em5.HmiInterface".cmTransferPnPLeftClampOpenClose.monitoring.inWorkPos;
               "HMI_Interface_Overview".homeCodition[5].emOverviewHomeLampOn[4] := "Unit1.Em5.HmiInterface".cmTransferPnPLeftJRDetect.monitoring.processValue;
               "HMI_Interface_Overview".homeCodition[5].emOverviewHomeLampOn[5] := FALSE;
               "HMI_Interface_Overview".homeCodition[5].emOverviewHomeLampOn[6] := FALSE;
               "HMI_Interface_Overview".homeCodition[5].emOverviewHomeLampOn[7] := FALSE;
               "HMI_Interface_Overview".homeCodition[5].emOverviewHomeLampOn[8] := FALSE;
               "HMI_Interface_Overview".homeCodition[5].emOverviewHomeLampOn[9] := FALSE;
               "HMI_Interface_Overview".homeCodition[5].emOverviewHomeLampOn[10] := FALSE;
               "HMI_Interface_Overview".homeCodition[5].emOverviewHomeLampOn[11] := FALSE;
               "HMI_Interface_Overview".homeCodition[5].emOverviewHomeLampOn[12] := FALSE;
               "HMI_Interface_Overview".homeCodition[5].emOverviewHomeLampOn[13] := FALSE;
           END_IF;
       END_IF;

       // Index 2
       IF "HMI_Interface_Overview".homeCodition[5].pageIndex = 2 THEN
           "HMI_Interface_Overview".homeCodition[5].emOverviewTitle := WSTRING#'P&P Right Home Condition 0';
           "HMI_Interface_Overview".homeCodition[5].emOverviewCmName[0] := WSTRING#'Transfer P&P Right X-Axis';
           "HMI_Interface_Overview".homeCodition[5].emOverviewCmName[1] := WSTRING#'Transfer P&P Right Y-Axis';
           "HMI_Interface_Overview".homeCodition[5].emOverviewCmName[2] := WSTRING#'Transfer P&P Right Z-Axis';
           "HMI_Interface_Overview".homeCodition[5].emOverviewCmName[3] := WSTRING#'Transfer P&P Right Clamp';
           "HMI_Interface_Overview".homeCodition[5].emOverviewCmName[4] := WSTRING#'Transfer P&P Right JR Detect';
           "HMI_Interface_Overview".homeCodition[5].emOverviewCmName[5] := WSTRING#'Spare';
           "HMI_Interface_Overview".homeCodition[5].emOverviewCmName[6] := WSTRING#'Spare';
           "HMI_Interface_Overview".homeCodition[5].emOverviewCmName[7] := WSTRING#'Spare';
           "HMI_Interface_Overview".homeCodition[5].emOverviewCmName[8] := WSTRING#'Spare';
           "HMI_Interface_Overview".homeCodition[5].emOverviewCmName[9] := WSTRING#'Spare';
           "HMI_Interface_Overview".homeCodition[5].emOverviewCmName[10] := WSTRING#'Spare';
           "HMI_Interface_Overview".homeCodition[5].emOverviewCmName[11] := WSTRING#'Spare';
           "HMI_Interface_Overview".homeCodition[5].emOverviewCmName[12] := WSTRING#'Spare';
           "HMI_Interface_Overview".homeCodition[5].emOverviewCmName[13] := WSTRING#'Spare';
           "HMI_Interface_Overview".homeCodition[5].emOverviewCmPositionName[0] := WSTRING#'Wait Position';
           "HMI_Interface_Overview".homeCodition[5].emOverviewCmPositionName[1] := WSTRING#'Wait Position';
           "HMI_Interface_Overview".homeCodition[5].emOverviewCmPositionName[2] := WSTRING#'Wait Position';
           "HMI_Interface_Overview".homeCodition[5].emOverviewCmPositionName[3] := WSTRING#'Open';
           "HMI_Interface_Overview".homeCodition[5].emOverviewCmPositionName[4] := WSTRING#'Not Detect';
           "HMI_Interface_Overview".homeCodition[5].emOverviewCmPositionName[5] := WSTRING#'Spare';
           "HMI_Interface_Overview".homeCodition[5].emOverviewCmPositionName[6] := WSTRING#'Spare';
           "HMI_Interface_Overview".homeCodition[5].emOverviewCmPositionName[7] := WSTRING#'Spare';
           "HMI_Interface_Overview".homeCodition[5].emOverviewCmPositionName[8] := WSTRING#'Spare';
           "HMI_Interface_Overview".homeCodition[5].emOverviewCmPositionName[9] := WSTRING#'Spare';
           "HMI_Interface_Overview".homeCodition[5].emOverviewCmPositionName[10] := WSTRING#'Spare';
           "HMI_Interface_Overview".homeCodition[5].emOverviewCmPositionName[11] := WSTRING#'Spare';
           "HMI_Interface_Overview".homeCodition[5].emOverviewCmPositionName[12] := WSTRING#'Spare';
           "HMI_Interface_Overview".homeCodition[5].emOverviewCmPositionName[13] := WSTRING#'Spare';
           IF NOT #statLampControl THEN
               "HMI_Interface_Overview".homeCodition[5].emOverviewHomeLampOn[0] := "Unit1.Em5.HmiInterface".cm.softcam.transferPnPRightAxisX.pos00_wait.inPos;
               "HMI_Interface_Overview".homeCodition[5].emOverviewHomeLampOn[1] := "Unit1.Em5.HmiInterface".cm.softcam.transferPnPRightAxisY.pos00_wait.inPos;
               "HMI_Interface_Overview".homeCodition[5].emOverviewHomeLampOn[2] := "Unit1.Em5.HmiInterface".cm.softcam.transferPnPRightAxisZ.pos00_wait.inPos;
               "HMI_Interface_Overview".homeCodition[5].emOverviewHomeLampOn[3] := "Unit1.Em5.HmiInterface".cmTransferPnPRightClampOpenClose.monitoring.inHomePos;
               "HMI_Interface_Overview".homeCodition[5].emOverviewHomeLampOn[4] := NOT "Unit1.Em5.HmiInterface".cmTransferPnPRightJRDetect.monitoring.processValue;
               "HMI_Interface_Overview".homeCodition[5].emOverviewHomeLampOn[5] := FALSE;
               "HMI_Interface_Overview".homeCodition[5].emOverviewHomeLampOn[6] := FALSE;
               "HMI_Interface_Overview".homeCodition[5].emOverviewHomeLampOn[7] := FALSE;
               "HMI_Interface_Overview".homeCodition[5].emOverviewHomeLampOn[8] := FALSE;
               "HMI_Interface_Overview".homeCodition[5].emOverviewHomeLampOn[9] := FALSE;
               "HMI_Interface_Overview".homeCodition[5].emOverviewHomeLampOn[10] := FALSE;
               "HMI_Interface_Overview".homeCodition[5].emOverviewHomeLampOn[11] := FALSE;
               "HMI_Interface_Overview".homeCodition[5].emOverviewHomeLampOn[12] := FALSE;
               "HMI_Interface_Overview".homeCodition[5].emOverviewHomeLampOn[13] := FALSE;
           END_IF;
       END_IF;

       // Index 3
       IF "HMI_Interface_Overview".homeCodition[5].pageIndex = 3 THEN
           "HMI_Interface_Overview".homeCodition[5].emOverviewTitle := WSTRING#'P&P Right Home Condition 1';
           "HMI_Interface_Overview".homeCodition[5].emOverviewCmName[0] := WSTRING#'Transfer P&P Right X-Axis';
           "HMI_Interface_Overview".homeCodition[5].emOverviewCmName[1] := WSTRING#'Transfer P&P Right Y-Axis';
           "HMI_Interface_Overview".homeCodition[5].emOverviewCmName[2] := WSTRING#'Transfer P&P Right Z-Axis';
           "HMI_Interface_Overview".homeCodition[5].emOverviewCmName[3] := WSTRING#'Transfer P&P Right Clamp';
           "HMI_Interface_Overview".homeCodition[5].emOverviewCmName[4] := WSTRING#'Transfer P&P Right JR Detect';
           "HMI_Interface_Overview".homeCodition[5].emOverviewCmName[5] := WSTRING#'Spare';
           "HMI_Interface_Overview".homeCodition[5].emOverviewCmName[6] := WSTRING#'Spare';
           "HMI_Interface_Overview".homeCodition[5].emOverviewCmName[7] := WSTRING#'Spare';
           "HMI_Interface_Overview".homeCodition[5].emOverviewCmName[8] := WSTRING#'Spare';
           "HMI_Interface_Overview".homeCodition[5].emOverviewCmName[9] := WSTRING#'Spare';
           "HMI_Interface_Overview".homeCodition[5].emOverviewCmName[10] := WSTRING#'Spare';
           "HMI_Interface_Overview".homeCodition[5].emOverviewCmName[11] := WSTRING#'Spare';
           "HMI_Interface_Overview".homeCodition[5].emOverviewCmName[12] := WSTRING#'Spare';
           "HMI_Interface_Overview".homeCodition[5].emOverviewCmName[13] := WSTRING#'Spare';
           "HMI_Interface_Overview".homeCodition[5].emOverviewCmPositionName[0] := WSTRING#'Wait Position';
           "HMI_Interface_Overview".homeCodition[5].emOverviewCmPositionName[1] := WSTRING#'Wait Position';
           "HMI_Interface_Overview".homeCodition[5].emOverviewCmPositionName[2] := WSTRING#'Wait Position';
           "HMI_Interface_Overview".homeCodition[5].emOverviewCmPositionName[3] := WSTRING#'Close';
           "HMI_Interface_Overview".homeCodition[5].emOverviewCmPositionName[4] := WSTRING#'Detect';
           "HMI_Interface_Overview".homeCodition[5].emOverviewCmPositionName[5] := WSTRING#'Spare';
           "HMI_Interface_Overview".homeCodition[5].emOverviewCmPositionName[6] := WSTRING#'Spare';
           "HMI_Interface_Overview".homeCodition[5].emOverviewCmPositionName[7] := WSTRING#'Spare';
           "HMI_Interface_Overview".homeCodition[5].emOverviewCmPositionName[8] := WSTRING#'Spare';
           "HMI_Interface_Overview".homeCodition[5].emOverviewCmPositionName[9] := WSTRING#'Spare';
           "HMI_Interface_Overview".homeCodition[5].emOverviewCmPositionName[10] := WSTRING#'Spare';
           "HMI_Interface_Overview".homeCodition[5].emOverviewCmPositionName[11] := WSTRING#'Spare';
           "HMI_Interface_Overview".homeCodition[5].emOverviewCmPositionName[12] := WSTRING#'Spare';
           "HMI_Interface_Overview".homeCodition[5].emOverviewCmPositionName[13] := WSTRING#'Spare';
           IF NOT #statLampControl THEN
               "HMI_Interface_Overview".homeCodition[5].emOverviewHomeLampOn[0] := "Unit1.Em5.HmiInterface".cm.softcam.transferPnPRightAxisX.pos00_wait.inPos;
               "HMI_Interface_Overview".homeCodition[5].emOverviewHomeLampOn[1] := "Unit1.Em5.HmiInterface".cm.softcam.transferPnPRightAxisY.pos00_wait.inPos;
               "HMI_Interface_Overview".homeCodition[5].emOverviewHomeLampOn[2] := "Unit1.Em5.HmiInterface".cm.softcam.transferPnPRightAxisZ.pos00_wait.inPos;
               "HMI_Interface_Overview".homeCodition[5].emOverviewHomeLampOn[3] := "Unit1.Em5.HmiInterface".cmTransferPnPRightClampOpenClose.monitoring.inWorkPos;
               "HMI_Interface_Overview".homeCodition[5].emOverviewHomeLampOn[4] := "Unit1.Em5.HmiInterface".cmTransferPnPRightJRDetect.monitoring.processValue;
               "HMI_Interface_Overview".homeCodition[5].emOverviewHomeLampOn[5] := FALSE;
               "HMI_Interface_Overview".homeCodition[5].emOverviewHomeLampOn[6] := FALSE;
               "HMI_Interface_Overview".homeCodition[5].emOverviewHomeLampOn[7] := FALSE;
               "HMI_Interface_Overview".homeCodition[5].emOverviewHomeLampOn[8] := FALSE;
               "HMI_Interface_Overview".homeCodition[5].emOverviewHomeLampOn[9] := FALSE;
               "HMI_Interface_Overview".homeCodition[5].emOverviewHomeLampOn[10] := FALSE;
               "HMI_Interface_Overview".homeCodition[5].emOverviewHomeLampOn[11] := FALSE;
               "HMI_Interface_Overview".homeCodition[5].emOverviewHomeLampOn[12] := FALSE;
               "HMI_Interface_Overview".homeCodition[5].emOverviewHomeLampOn[13] := FALSE;
           END_IF;
       END_IF;

   END_REGION
END_REGION

REGION Network 36 (SCL): Em 6 Page Index Mapping
   REGION Page Index

       // Index 0
       IF "HMI_Interface_Overview".homeCodition[6].pageIndex = 0 THEN
           "HMI_Interface_Overview".homeCodition[6].emOverviewTitle := WSTRING#'Home Condition 0';
           "HMI_Interface_Overview".homeCodition[6].emOverviewCmName[0] := WSTRING#'Hot Press Left Servo Press';
           "HMI_Interface_Overview".homeCodition[6].emOverviewCmName[1] := WSTRING#'Hot Press Left Stage Lift Front';
           "HMI_Interface_Overview".homeCodition[6].emOverviewCmName[2] := WSTRING#'Hot Press Left Stage Lift Rear';
           "HMI_Interface_Overview".homeCodition[6].emOverviewCmName[3] := WSTRING#'Hot Press Left JR Detect';
           "HMI_Interface_Overview".homeCodition[6].emOverviewCmName[4] := WSTRING#'Spare';
           "HMI_Interface_Overview".homeCodition[6].emOverviewCmName[5] := WSTRING#'Spare';
           "HMI_Interface_Overview".homeCodition[6].emOverviewCmName[6] := WSTRING#'Spare';
           "HMI_Interface_Overview".homeCodition[6].emOverviewCmName[7] := WSTRING#'Spare';
           "HMI_Interface_Overview".homeCodition[6].emOverviewCmName[8] := WSTRING#'Spare';
           "HMI_Interface_Overview".homeCodition[6].emOverviewCmName[9] := WSTRING#'Spare';
           "HMI_Interface_Overview".homeCodition[6].emOverviewCmName[10] := WSTRING#'Spare';
           "HMI_Interface_Overview".homeCodition[6].emOverviewCmName[11] := WSTRING#'Spare';
           "HMI_Interface_Overview".homeCodition[6].emOverviewCmName[12] := WSTRING#'Spare';
           "HMI_Interface_Overview".homeCodition[6].emOverviewCmName[13] := WSTRING#'Spare';
           "HMI_Interface_Overview".homeCodition[6].emOverviewCmPositionName[0] := WSTRING#'Home Position';
           "HMI_Interface_Overview".homeCodition[6].emOverviewCmPositionName[1] := WSTRING#'Down';
           "HMI_Interface_Overview".homeCodition[6].emOverviewCmPositionName[2] := WSTRING#'Down';
           "HMI_Interface_Overview".homeCodition[6].emOverviewCmPositionName[3] := WSTRING#'Not Detect';
           "HMI_Interface_Overview".homeCodition[6].emOverviewCmPositionName[4] := WSTRING#'Spare';
           "HMI_Interface_Overview".homeCodition[6].emOverviewCmPositionName[5] := WSTRING#'Spare';
           "HMI_Interface_Overview".homeCodition[6].emOverviewCmPositionName[6] := WSTRING#'Spare';
           "HMI_Interface_Overview".homeCodition[6].emOverviewCmPositionName[7] := WSTRING#'Spare';
           "HMI_Interface_Overview".homeCodition[6].emOverviewCmPositionName[8] := WSTRING#'Spare';
           "HMI_Interface_Overview".homeCodition[6].emOverviewCmPositionName[9] := WSTRING#'Spare';
           "HMI_Interface_Overview".homeCodition[6].emOverviewCmPositionName[10] := WSTRING#'Spare';
           "HMI_Interface_Overview".homeCodition[6].emOverviewCmPositionName[11] := WSTRING#'Spare';
           "HMI_Interface_Overview".homeCodition[6].emOverviewCmPositionName[12] := WSTRING#'Spare';
           "HMI_Interface_Overview".homeCodition[6].emOverviewCmPositionName[13] := WSTRING#'Spare';
           IF NOT #statLampControl THEN
               "HMI_Interface_Overview".homeCodition[6].emOverviewHomeLampOn[0] := "Unit1.Em6.HmiInterface".cmHotPressLeftServoPress.monitoring.profinetInput."HOME-POS-REACHED";
               "HMI_Interface_Overview".homeCodition[6].emOverviewHomeLampOn[1] := "Unit1.Em6.HmiInterface".cmHotpressLeftStageLiftFrontUpDown.monitoring.inWorkPos;
               "HMI_Interface_Overview".homeCodition[6].emOverviewHomeLampOn[2] := "Unit1.Em6.HmiInterface".cmHotpressLeftStageLiftRearUpDown.monitoring.inWorkPos;
               "HMI_Interface_Overview".homeCodition[6].emOverviewHomeLampOn[3] := NOT "Unit1.Em6.HmiInterface".cmHotpressLeftJRDetect.monitoring.processValue;
               "HMI_Interface_Overview".homeCodition[6].emOverviewHomeLampOn[4] := FALSE;
               "HMI_Interface_Overview".homeCodition[6].emOverviewHomeLampOn[5] := FALSE;
               "HMI_Interface_Overview".homeCodition[6].emOverviewHomeLampOn[6] := FALSE;
               "HMI_Interface_Overview".homeCodition[6].emOverviewHomeLampOn[7] := FALSE;
               "HMI_Interface_Overview".homeCodition[6].emOverviewHomeLampOn[8] := FALSE;
               "HMI_Interface_Overview".homeCodition[6].emOverviewHomeLampOn[9] := FALSE;
               "HMI_Interface_Overview".homeCodition[6].emOverviewHomeLampOn[10] := FALSE;
               "HMI_Interface_Overview".homeCodition[6].emOverviewHomeLampOn[11] := FALSE;
               "HMI_Interface_Overview".homeCodition[6].emOverviewHomeLampOn[12] := FALSE;
               "HMI_Interface_Overview".homeCodition[6].emOverviewHomeLampOn[13] := FALSE;
           END_IF;
       END_IF;

       // Index 1
       IF "HMI_Interface_Overview".homeCodition[6].pageIndex = 1 THEN
           "HMI_Interface_Overview".homeCodition[6].emOverviewTitle := WSTRING#'Home Condition 1';
           "HMI_Interface_Overview".homeCodition[6].emOverviewCmName[0] := WSTRING#'Hot Press Left Servo Press';
           "HMI_Interface_Overview".homeCodition[6].emOverviewCmName[1] := WSTRING#'Hot Press Left Stage Lift Front';
           "HMI_Interface_Overview".homeCodition[6].emOverviewCmName[2] := WSTRING#'Hot Press Left Stage Lift Rear';
           "HMI_Interface_Overview".homeCodition[6].emOverviewCmName[3] := WSTRING#'Hot Press Left JR Detect';
           "HMI_Interface_Overview".homeCodition[6].emOverviewCmName[4] := WSTRING#'Spare';
           "HMI_Interface_Overview".homeCodition[6].emOverviewCmName[5] := WSTRING#'Spare';
           "HMI_Interface_Overview".homeCodition[6].emOverviewCmName[6] := WSTRING#'Spare';
           "HMI_Interface_Overview".homeCodition[6].emOverviewCmName[7] := WSTRING#'Spare';
           "HMI_Interface_Overview".homeCodition[6].emOverviewCmName[8] := WSTRING#'Spare';
           "HMI_Interface_Overview".homeCodition[6].emOverviewCmName[9] := WSTRING#'Spare';
           "HMI_Interface_Overview".homeCodition[6].emOverviewCmName[10] := WSTRING#'Spare';
           "HMI_Interface_Overview".homeCodition[6].emOverviewCmName[11] := WSTRING#'Spare';
           "HMI_Interface_Overview".homeCodition[6].emOverviewCmName[12] := WSTRING#'Spare';
           "HMI_Interface_Overview".homeCodition[6].emOverviewCmName[13] := WSTRING#'Spare';
           "HMI_Interface_Overview".homeCodition[6].emOverviewCmPositionName[0] := WSTRING#'Home Position';
           "HMI_Interface_Overview".homeCodition[6].emOverviewCmPositionName[1] := WSTRING#'Down';
           "HMI_Interface_Overview".homeCodition[6].emOverviewCmPositionName[2] := WSTRING#'Down';
           "HMI_Interface_Overview".homeCodition[6].emOverviewCmPositionName[3] := WSTRING#'Detect';
           "HMI_Interface_Overview".homeCodition[6].emOverviewCmPositionName[4] := WSTRING#'Spare';
           "HMI_Interface_Overview".homeCodition[6].emOverviewCmPositionName[5] := WSTRING#'Spare';
           "HMI_Interface_Overview".homeCodition[6].emOverviewCmPositionName[6] := WSTRING#'Spare';
           "HMI_Interface_Overview".homeCodition[6].emOverviewCmPositionName[7] := WSTRING#'Spare';
           "HMI_Interface_Overview".homeCodition[6].emOverviewCmPositionName[8] := WSTRING#'Spare';
           "HMI_Interface_Overview".homeCodition[6].emOverviewCmPositionName[9] := WSTRING#'Spare';
           "HMI_Interface_Overview".homeCodition[6].emOverviewCmPositionName[10] := WSTRING#'Spare';
           "HMI_Interface_Overview".homeCodition[6].emOverviewCmPositionName[11] := WSTRING#'Spare';
           "HMI_Interface_Overview".homeCodition[6].emOverviewCmPositionName[12] := WSTRING#'Spare';
           "HMI_Interface_Overview".homeCodition[6].emOverviewCmPositionName[13] := WSTRING#'Spare';
           IF NOT #statLampControl THEN
               "HMI_Interface_Overview".homeCodition[6].emOverviewHomeLampOn[0] := "Unit1.Em6.HmiInterface".cmHotPressLeftServoPress.monitoring.profinetInput."HOME-POS-REACHED";
               "HMI_Interface_Overview".homeCodition[6].emOverviewHomeLampOn[1] := "Unit1.Em6.HmiInterface".cmHotpressLeftStageLiftFrontUpDown.monitoring.inWorkPos;
               "HMI_Interface_Overview".homeCodition[6].emOverviewHomeLampOn[2] := "Unit1.Em6.HmiInterface".cmHotpressLeftStageLiftRearUpDown.monitoring.inWorkPos;
               "HMI_Interface_Overview".homeCodition[6].emOverviewHomeLampOn[3] := "Unit1.Em6.HmiInterface".cmHotpressLeftJRDetect.monitoring.processValue;
               "HMI_Interface_Overview".homeCodition[6].emOverviewHomeLampOn[4] := FALSE;
               "HMI_Interface_Overview".homeCodition[6].emOverviewHomeLampOn[5] := FALSE;
               "HMI_Interface_Overview".homeCodition[6].emOverviewHomeLampOn[6] := FALSE;
               "HMI_Interface_Overview".homeCodition[6].emOverviewHomeLampOn[7] := FALSE;
               "HMI_Interface_Overview".homeCodition[6].emOverviewHomeLampOn[8] := FALSE;
               "HMI_Interface_Overview".homeCodition[6].emOverviewHomeLampOn[9] := FALSE;
               "HMI_Interface_Overview".homeCodition[6].emOverviewHomeLampOn[10] := FALSE;
               "HMI_Interface_Overview".homeCodition[6].emOverviewHomeLampOn[11] := FALSE;
               "HMI_Interface_Overview".homeCodition[6].emOverviewHomeLampOn[12] := FALSE;
               "HMI_Interface_Overview".homeCodition[6].emOverviewHomeLampOn[13] := FALSE;
           END_IF;
       END_IF;

   END_REGION
END_REGION

REGION Network 37 (SCL): Em 7 Page Index Mapping
   REGION Page Index

       // Index 0
       IF "HMI_Interface_Overview".homeCodition[7].pageIndex = 0 THEN
           "HMI_Interface_Overview".homeCodition[7].emOverviewTitle := WSTRING#'Home Condition 0';
           "HMI_Interface_Overview".homeCodition[7].emOverviewCmName[0] := WSTRING#'Hot Press Right Servo Press';
           "HMI_Interface_Overview".homeCodition[7].emOverviewCmName[1] := WSTRING#'Hot Press Right Stage Lift Front';
           "HMI_Interface_Overview".homeCodition[7].emOverviewCmName[2] := WSTRING#'Hot Press Right Stage Lift Rear';
           "HMI_Interface_Overview".homeCodition[7].emOverviewCmName[3] := WSTRING#'Hot Press Right JR Detect';
           "HMI_Interface_Overview".homeCodition[7].emOverviewCmName[4] := WSTRING#'Spare';
           "HMI_Interface_Overview".homeCodition[7].emOverviewCmName[5] := WSTRING#'Spare';
           "HMI_Interface_Overview".homeCodition[7].emOverviewCmName[6] := WSTRING#'Spare';
           "HMI_Interface_Overview".homeCodition[7].emOverviewCmName[7] := WSTRING#'Spare';
           "HMI_Interface_Overview".homeCodition[7].emOverviewCmName[8] := WSTRING#'Spare';
           "HMI_Interface_Overview".homeCodition[7].emOverviewCmName[9] := WSTRING#'Spare';
           "HMI_Interface_Overview".homeCodition[7].emOverviewCmName[10] := WSTRING#'Spare';
           "HMI_Interface_Overview".homeCodition[7].emOverviewCmName[11] := WSTRING#'Spare';
           "HMI_Interface_Overview".homeCodition[7].emOverviewCmName[12] := WSTRING#'Spare';
           "HMI_Interface_Overview".homeCodition[7].emOverviewCmName[13] := WSTRING#'Spare';
           "HMI_Interface_Overview".homeCodition[7].emOverviewCmPositionName[0] := WSTRING#'Home Position';
           "HMI_Interface_Overview".homeCodition[7].emOverviewCmPositionName[1] := WSTRING#'Down';
           "HMI_Interface_Overview".homeCodition[7].emOverviewCmPositionName[2] := WSTRING#'Down';
           "HMI_Interface_Overview".homeCodition[7].emOverviewCmPositionName[3] := WSTRING#'Not Detect';
           "HMI_Interface_Overview".homeCodition[7].emOverviewCmPositionName[4] := WSTRING#'Spare';
           "HMI_Interface_Overview".homeCodition[7].emOverviewCmPositionName[5] := WSTRING#'Spare';
           "HMI_Interface_Overview".homeCodition[7].emOverviewCmPositionName[6] := WSTRING#'Spare';
           "HMI_Interface_Overview".homeCodition[7].emOverviewCmPositionName[7] := WSTRING#'Spare';
           "HMI_Interface_Overview".homeCodition[7].emOverviewCmPositionName[8] := WSTRING#'Spare';
           "HMI_Interface_Overview".homeCodition[7].emOverviewCmPositionName[9] := WSTRING#'Spare';
           "HMI_Interface_Overview".homeCodition[7].emOverviewCmPositionName[10] := WSTRING#'Spare';
           "HMI_Interface_Overview".homeCodition[7].emOverviewCmPositionName[11] := WSTRING#'Spare';
           "HMI_Interface_Overview".homeCodition[7].emOverviewCmPositionName[12] := WSTRING#'Spare';
           "HMI_Interface_Overview".homeCodition[7].emOverviewCmPositionName[13] := WSTRING#'Spare';
           IF NOT #statLampControl THEN
               "HMI_Interface_Overview".homeCodition[7].emOverviewHomeLampOn[0] := "Unit1.Em7.HmiInterface".cmHotPressRightServoPress.monitoring.profinetInput."HOME-POS-REACHED";
               "HMI_Interface_Overview".homeCodition[7].emOverviewHomeLampOn[1] := "Unit1.Em7.HmiInterface".cmHotPressRightStageLiftFrontUpDown.monitoring.inWorkPos;
               "HMI_Interface_Overview".homeCodition[7].emOverviewHomeLampOn[2] := "Unit1.Em7.HmiInterface".cmHotPressRightStageLiftRearUpDown.monitoring.inWorkPos;
               "HMI_Interface_Overview".homeCodition[7].emOverviewHomeLampOn[3] := NOT "Unit1.Em7.HmiInterface".cmHotPressRightJRDetect.monitoring.processValue;
               "HMI_Interface_Overview".homeCodition[7].emOverviewHomeLampOn[4] := FALSE;
               "HMI_Interface_Overview".homeCodition[7].emOverviewHomeLampOn[5] := FALSE;
               "HMI_Interface_Overview".homeCodition[7].emOverviewHomeLampOn[6] := FALSE;
               "HMI_Interface_Overview".homeCodition[7].emOverviewHomeLampOn[7] := FALSE;
               "HMI_Interface_Overview".homeCodition[7].emOverviewHomeLampOn[8] := FALSE;
               "HMI_Interface_Overview".homeCodition[7].emOverviewHomeLampOn[9] := FALSE;
               "HMI_Interface_Overview".homeCodition[7].emOverviewHomeLampOn[10] := FALSE;
               "HMI_Interface_Overview".homeCodition[7].emOverviewHomeLampOn[11] := FALSE;
               "HMI_Interface_Overview".homeCodition[7].emOverviewHomeLampOn[12] := FALSE;
               "HMI_Interface_Overview".homeCodition[7].emOverviewHomeLampOn[13] := FALSE;
           END_IF;
       END_IF;

